# B&R Automation Studio project RTFProj (part 2)

#### measurement_ofScore.c
```c
#include <bur/plctypes.h>
#include <bur/plc.h>
#include <astime.h>
#include <string.h>
#include <math.h>

#ifdef __cplusplus
	extern "C"
	{
#endif
	#include "rp_funcx1.h"
#ifdef __cplusplus
	};
#endif
void initialization(struct measurement_ofScore* m_oS);

void measurement_ofScore(struct measurement_ofScore* m_oS)
{

    if(!m_oS->Enable){
        initialization(m_oS);
    }

    switch(m_oS->Internal.state){
        case 0:
            {
                if(m_oS->Internal.counter <= 0){
                    m_oS->Internal.counter = 0;
                }

                m_oS->Internal.results[0]   = strcmp(m_oS->PLAYER1_NAME, "");
                m_oS->Internal.results[1]   = strcmp(m_oS->PLAYER2_NAME, "");

                if(m_oS->start_measurement == 1 && m_oS->Error == 0){
                    if(m_oS->Internal.results[0] == 0 && m_oS->Internal.results[1] == 0){
                        m_oS->Internal.auxiliary_str[5] = (UDINT) strcpy(m_oS->PLAYER1_NAME,"PLAYER 1");
                        m_oS->Internal.auxiliary_str[6] = (UDINT) strcpy(m_oS->PLAYER2_NAME,"PLAYER 2");
                    }
                    // CPU NAME
                    m_oS->Internal.auxiliary_str[7] = (UDINT) strcpy(m_oS->team_nameCPU,"B&R ROBOT");
                    // HUMAN NAME
                    strcpy(m_oS->Internal.string[5],m_oS->PLAYER1_NAME);
                    strcpy(m_oS->Internal.string[6]," \n \t& \n");
                    strcpy(m_oS->Internal.string[8], m_oS->PLAYER2_NAME);
                    m_oS->Internal.auxiliary_str[8] = (UDINT) strcat(m_oS->Internal.string[5], m_oS->Internal.string[6]);
                    strcpy(m_oS->Internal.string[7], m_oS->Internal.string[5]);
                    m_oS->Internal.auxiliary_str[9] = (UDINT) strcat(m_oS->Internal.string[7], m_oS->Internal.string[8]);
                    m_oS->Internal.auxiliary_str[10] = (UDINT) strcpy(m_oS->team_nameHUM,m_oS->Internal.auxiliary_str[9]);
                    // CHANGE STATE
                    m_oS->Internal.state = 1;
                }else if(m_oS->Error == 1){
                    m_oS->Internal.state = 5;
                }else if(m_oS->pause == 1){
                    m_oS->Internal.before_state = m_oS->Internal.state;
                    m_oS->Internal.state = 6;
                }else{
                    m_oS->Internal.state = 0;
                }
            }
            break;
        case 1:
            {
                if(m_oS->sens_wicket_CPU == 1){
                    m_oS->count_goals_CPU++;
                    m_oS->sens_wicket_CPU = 0;
                }

                if(m_oS->sens_wicket_HUM == 1){
                    m_oS->count_goals_HUM++;
                    m_oS->sens_wicket_HUM = 0;
                }

                if((m_oS->count_goals_HUM - m_oS->count_goals_CPU) == 0){
                    m_oS->probability_CPU = 50;
                    m_oS->probability_HUM = 50;
                }else if((m_oS->count_goals_HUM - m_oS->count_goals_CPU) < 0){
                    if(fabs((m_oS->count_goals_HUM - m_oS->count_goals_CPU)) <= 5){
                        m_oS->probability_CPU = 50 + fabs((m_oS->count_goals_HUM - m_oS->count_goals_CPU))*10;
                        m_oS->probability_HUM = 100 - m_oS->probability_CPU;
                    }else{
                        m_oS->probability_CPU = 100;
                        m_oS->probability_HUM = 0;
                    }
                }else{
                    if(fabs((m_oS->count_goals_HUM - m_oS->count_goals_CPU)) <= 5){
                        m_oS->probability_HUM = 50 + fabs((m_oS->count_goals_HUM - m_oS->count_goals_CPU))*10;
                        m_oS->probability_CPU = 100 - m_oS->probability_HUM;
                    }else{
                        m_oS->probability_HUM = 100;
                        m_oS->probability_CPU = 0;
                    }
                }
				if(((m_oS->count_goals_CPU + m_oS->count_goals_HUM) == 10) && m_oS->Error == 0){
					if(m_oS->count_goals_CPU > m_oS->count_goals_HUM){
						m_oS->Internal.WINNER++;
					}else if(m_oS->count_goals_CPU == m_oS->count_goals_HUM){
						m_oS->Internal.DRAW++;
					}else if(m_oS->count_goals_CPU < m_oS->count_goals_HUM){
						m_oS->Internal.LOSE++;
					}
					// change state
					m_oS->Internal.state             = 2;
					m_oS->Internal.write_matchInfo   = 1;
				}else if(m_oS->exit_game == 1 ){
                    m_oS->Internal.state = 3;
                }else if(m_oS->restart_measurement == 1){
                    m_oS->Internal.state = 4;
                }else if(m_oS->Error == 1){
                    m_oS->Internal.state = 5;
                }else if(m_oS->pause == 1){
                    m_oS->Internal.before_state = m_oS->Internal.state;
                    m_oS->Internal.state = 6;
                }else{
                    m_oS->Internal.state = 1;
                }

            }
            break;
        case 2:
            {
                if(m_oS->Internal.write_matchInfo == 1){
                    // call FB : Get time and date
                    m_oS->Internal.UtcDTStructureGetTime_1.enable = 1;
                    m_oS->Internal.UtcDTStructureGetTime_1.pDTStructure = (UDINT) &m_oS->Internal.DTStruct;
                    UtcDTStructureGetTime(&m_oS->Internal.UtcDTStructureGetTime_1);
                    ascDTStructure((UDINT) &m_oS->Internal.DTStruct, (UDINT) &m_oS->Internal.string[0], m_oS->Internal.length);
                    // write time and date into the variable
                    m_oS->Internal.auxiliary_str[0] = (UDINT) strcpy(m_oS->match_informations.date[m_oS->Internal.counter],m_oS->Internal.string[0]);
                    // write score
                    m_oS->match_informations.score_CPU[m_oS->Internal.counter] = m_oS->count_goals_CPU;
                    m_oS->match_informations.score_HUM[m_oS->Internal.counter] = m_oS->count_goals_HUM;
                    // write name of B&R team
                    m_oS->Internal.auxiliary_str[1] = (UDINT) strcpy(m_oS->match_informations.team_name_CPU[m_oS->Internal.counter],"B&R ROBOT");
                    // write names of both players
                    strcpy(m_oS->Internal.string[1],m_oS->PLAYER1_NAME);
                    strcpy(m_oS->Internal.string[2]," & ");
                    strcpy(m_oS->Internal.string[4], m_oS->PLAYER2_NAME);
                    m_oS->Internal.auxiliary_str[2] = (UDINT) strcat(m_oS->Internal.string[1], m_oS->Internal.string[2]);
                    strcpy(m_oS->Internal.string[3], m_oS->Internal.string[1]);
                    m_oS->Internal.auxiliary_str[3] = (UDINT) strcat(m_oS->Internal.string[3], m_oS->Internal.string[4]);
                    m_oS->Internal.auxiliary_str[4] = (UDINT) strcpy(m_oS->match_informations.team_name_HUM[m_oS->Internal.counter],m_oS->Internal.auxiliary_str[3]);

                    m_oS->Internal.counter++;
                    m_oS->Internal.write_matchInfo = 0;
                }

                if(m_oS->exit_game == 1){
                    m_oS->Internal.state = 3;
                }else if(m_oS->restart_measurement == 1){
                    m_oS->Internal.state = 4;
                }else if(m_oS->Error == 1){
                    m_oS->Internal.state = 5;
                }else if(m_oS->pause == 1){
                    m_oS->Internal.before_state = m_oS->Internal.state;
                    m_oS->Internal.state = 6;
                }else{
                    m_oS->Internal.state = 2;
                }
            }
            break;
        case 3:
            {
                // exit game
                m_oS->start_measurement   = 0;
                m_oS->exit_game           = 0;
                m_oS->restart_measurement = 0;
                m_oS->count_goals_CPU     = 0;
                m_oS->count_goals_HUM     = 0;

                m_oS->Internal.e_r_str[0] = (UDINT) strcpy(m_oS->PLAYER1_NAME,"");
                m_oS->Internal.e_r_str[1] = (UDINT) strcpy(m_oS->PLAYER2_NAME,"");

                if(m_oS->Error == 1){
                    m_oS->Internal.state = 5;
                }else if(m_oS->pause == 1){
                    m_oS->Internal.before_state = m_oS->Internal.state;
                    m_oS->Internal.state = 6;
                }else{
                    m_oS->Internal.state = 0;
                }
            }
            break;
        case 4:
            {
                // restart game
                m_oS->start_measurement   = 0;
                m_oS->exit_game           = 0;
                m_oS->restart_measurement = 0;
                m_oS->count_goals_CPU     = 0;
                m_oS->count_goals_HUM     = 0;

                m_oS->Internal.e_r_str[2] = (UDINT) strcpy(m_oS->PLAYER1_NAME,m_oS->PLAYER1_NAME);
                m_oS->Internal.e_r_str[3] = (UDINT) strcpy(m_oS->PLAYER2_NAME,m_oS->PLAYER2_NAME);

                if(m_oS->Error == 1){
                    m_oS->Internal.state = 5;
                }else if(m_oS->pause == 1){
                    m_oS->Internal.before_state = m_oS->Internal.state;
                    m_oS->Internal.state = 6;
                }else{
                    m_oS->Internal.state = 1;
                }
            }
            break;
        case 5:
            {
                // error state
                if(m_oS->Error == 0){
                    m_oS->Internal.state = 3;
                }else if(m_oS->pause == 1){
                    m_oS->Internal.before_state = m_oS->Internal.state;
                    m_oS->Internal.state = 6;
                }
            }
            break;
        case 6:
            {
                // pause
                if(m_oS->Error == 1){
                    m_oS->Internal.state = 5;
                }else if(m_oS->pause == 0){
                    m_oS->Internal.state = m_oS->Internal.before_state;
                }
            }
            break;
    }// end switch

}// end fucntion

void initialization(struct measurement_ofScore* m_oS){
    m_oS->Internal.state             = 0;
    m_oS->Internal.e_r_str[0]        = 0;
    m_oS->Internal.e_r_str[1]        = 0;
    m_oS->Internal.e_r_str[2]        = 0;
    m_oS->Internal.e_r_str[3]        = 0;
    m_oS->Internal.auxiliary_str[0]  = 0;
    m_oS->Internal.auxiliary_str[1]  = 0;
    m_oS->Internal.auxiliary_str[2]  = 0;
    m_oS->Internal.auxiliary_str[3]  = 0;
    m_oS->Internal.auxiliary_str[4]  = 0;
    m_oS->Internal.auxiliary_str[5]  = 0;
    m_oS->Internal.auxiliary_str[6]  = 0;
    m_oS->Internal.auxiliary_str[7]  = 0;
    m_oS->Internal.auxiliary_str[8]  = 0;
    m_oS->Internal.auxiliary_str[9]  = 0;
    m_oS->Internal.auxiliary_str[10] = 0;
    m_oS->Internal.counter           = 0;
    m_oS->Internal.length            = 25;
    m_oS->Internal.write_matchInfo   = 0;
    m_oS->Internal.results[0]        = 0;
    m_oS->Internal.results[1]        = 0;
	m_oS->Internal.before_state      = 0;
	m_oS->Internal.WINNER			 = 0;
	m_oS->Internal.DRAW			     = 0;
	m_oS->Internal.LOSE				 = 0;
    m_oS->count_goals_CPU            = 0;
    m_oS->count_goals_HUM            = 0;
    m_oS->sens_wicket_HUM            = 0;
    m_oS->restart_measurement        = 0;
    m_oS->pause                      = 0;
    m_oS->exit_game                  = 0;
    m_oS->start_measurement          = 0;
    m_oS->probability_CPU            = 50;
    m_oS->probability_HUM            = 50;
}// end function
```

#### start_linearAxis.c
```c
#include <bur/plctypes.h>
#include <stdio.h>
#include <stdlib.h>
#include <MpAxis.h>

#ifdef __cplusplus
	extern "C"
	{
#endif
	#include "rp_funcx1.h"
#ifdef __cplusplus
	};
#endif
void initialization_sla(struct start_linearAxis* s_la);

void start_linearAxis(struct start_linearAxis* s_la)
{
	if(!s_la->Enable){
		initialization_sla(s_la);
	}

	switch(s_la->Internal.state){
		case 0:
			{
				s_la->Internal.before_state     = s_la->Internal.state;

				if(s_la->start_btn == 1){
					// adjustment parameters -> axis
					s_la->axis_param->Home.Mode 				  = mpAXIS_HOME_MODE_BLOCK_TORQUE;
					s_la->axis_param->Home.Position 		  	  = s_la->max_leftPosition;
					s_la->axis_param->Home.StartVelocity   		  = s_la->velocity;
					s_la->axis_param->Home.HomingVelocity  		  = s_la->velocity;
					s_la->axis_param->Home.Acceleration    		  = 200000;
					s_la->axis_param->Home.StartDirection  		  = mpAXIS_HOME_DIR_POSITIVE;
					s_la->axis_param->Home.HomingDirection 		  = mpAXIS_HOME_DIR_NEGATIVE;
					s_la->axis_param->Home.TorqueLimit	 		  = 0.02;
					s_la->axis_param->Home.PositionErrorStopLimit = s_la->max_leftPosition + 10;
					// reset output
					s_la->succesfully = 0;
					if(s_la->axis_name->Error == 1 || s_la->axis_name->StatusID != 0){
						s_la->axis_name->ErrorReset = 0;
						if(s_la->axis_name->ErrorReset == 0){
							s_la->Internal.state = 10;
						}
					}else{
						if(s_la->start_btn == 1){
							s_la->Internal.state = 1;
						}
					}
				}
			}
			break;
		case 1:
			{
				s_la->Internal.before_state = s_la->Internal.state;
				// power on -> axis
				s_la->axis_name->Power = 1;

				if(s_la->axis_name->Error == 1 || s_la->axis_name->StatusID != 0){
					s_la->axis_name->ErrorReset = 0;
					if(s_la->axis_name->ErrorReset == 0){
						s_la->Internal.state = 10;
					}
				}else{
					if(s_la->axis_name->PowerOn == 1){
						s_la->Internal.state = 2;
					}
				}
			}
			break;
		case 2:
			{
				s_la->Internal.before_state = s_la->Internal.state;
				// update -> axis
				s_la->axis_name->Update = 1;

				if(s_la->axis_name->Error == 1 || s_la->axis_name->StatusID != 0){
					s_la->axis_name->ErrorReset = 0;
					if(s_la->axis_name->ErrorReset == 0){
						s_la->Internal.state = 10;
					}
				}else{
					if(s_la->axis_name->UpdateDone == 1){
						s_la->axis_name->Update = 0;
						if(s_la->axis_name->UpdateDone == 0){
							s_la->Internal.state 	= 3;
						}
					}
				}
			}
		case 3:
			{
				s_la->Internal.before_state = s_la->Internal.state;
				// home -> axis
				s_la->axis_name->Home = 1;

				if(s_la->axis_name->Error == 1 || s_la->axis_name->StatusID != 0){
					s_la->axis_name->ErrorReset = 0;
					if(s_la->axis_name->ErrorReset == 0){
						s_la->Internal.state = 10;
					}
				}else{
					if(s_la->axis_name->IsHomed == 1){
						s_la->axis_name->Home = 0;
						s_la->succesfully     = 1;
						s_la->Internal.state  = 0;
					}
				}
			}
			break;
		case 10:
			{
				s_la->axis_name->ErrorReset = 1;

				if(s_la->axis_name->Error == 1 || s_la->axis_name->StatusID != 0){
					s_la->Internal.state = 10;
				}else{
					s_la->axis_name->ErrorReset = 0;
					s_la->Internal.state 		= s_la->Internal.before_state;
				}
			}
			break;
	}// end switch
}// end function

void initialization_sla(struct start_linearAxis* s_la)
{
	s_la->Internal.state 		= 0;
	s_la->Internal.before_state = 0;
	s_la->start_btn				= 0;
	s_la->succesfully     		= 0;
}// end function
```

#### start_virtualAxis.c
```c
#include <bur/plctypes.h>
#include <stdio.h>
#include <stdlib.h>
#include <MpAxis.h>

#ifdef __cplusplus
	extern "C"
	{
#endif
	#include "rp_funcx1.h"
#ifdef __cplusplus
	};
#endif
void initialization_sva(struct start_virtualAxis* s_va);

void start_virtualAxis(struct start_virtualAxis* s_va)
{
	if(!s_va->Enable){
		initialization_sra(s_va);
	}

	switch(s_va->Internal.state){
		case 0:
			{
				s_va->Internal.before_state     = s_va->Internal.state;

				if(s_va->start_btn == 1){
					// reset output {virtual}
					s_va->succesfully = 0;
					if(s_va->axis_name->Error == 1 || s_va->axis_name->StatusID != 0){
						s_va->axis_name->ErrorReset = 0;
						if(s_va->axis_name->ErrorReset == 0){
							s_va->Internal.state = 10;
						}
					}else{
						if(s_va->start_btn == 1){
							s_va->Internal.state = 1;
						}
					}
				}
			}
			break;
		case 1:
			{
				s_va->Internal.before_state = s_va->Internal.state;
				// power on -> axis
				s_va->axis_name->Power = 1;

				if(s_va->axis_name->Error == 1 || s_va->axis_name->StatusID != 0){
					s_va->axis_name->ErrorReset = 0;
					if(s_va->axis_name->ErrorReset == 0){
						s_va->Internal.state = 10;
					}
				}else{
					if(s_va->axis_name->PowerOn == 1){
						s_va->Internal.state = 2;
					}
				}
			}
			break;
		case 2:
			{
				s_va->Internal.before_state = s_va->Internal.state;
				// home -> axis
				s_va->axis_name->Home = 1;

				if(s_va->axis_name->Error == 1 || s_va->axis_name->StatusID != 0){
					s_va->axis_name->ErrorReset = 0;
					if(s_va->axis_name->ErrorReset == 0){
						s_va->Internal.state = 10;
					}
				}else{
					if(s_va->axis_name->IsHomed == 1){
						s_va->axis_name->Home = 0;
						s_va->Internal.state  = 3;
					}
				}
			}
			break;
		case 3:
			{
				s_va->Internal.before_state = s_va->Internal.state;

				if(s_va->axis_name->Error == 1 || s_va->axis_name->StatusID != 0){
					s_va->axis_name->ErrorReset = 0;
					if(s_va->axis_name->ErrorReset == 0){
						s_va->Internal.state = 10;
					}
				}else{
					s_va->succesfully	 = 1;
					s_va->Internal.state = 0;
				}
			}
			break;
		case 10:
			{
				s_va->axis_name->ErrorReset = 1;

				if(s_va->axis_name->Error == 1 || s_va->axis_name->StatusID != 0){
					s_va->Internal.state = 10;
				}else{
					s_va->axis_name->ErrorReset = 0;
					s_va->Internal.state 		= s_va->Internal.before_state;
				}
			}
			break;
	}// end switch
}// end function

void initialization_sva(struct start_virtualAxis* s_va)
{
	s_va->Internal.state 		= 0;
	s_va->Internal.before_state = 0;
	s_va->start_btn				= 0;
	s_va->succesfully     		= 0;
}// end function
```

#### start_rotaryAxis.c
```c
#include <bur/plctypes.h>
#include <stdio.h>
#include <stdlib.h>
#include <MpAxis.h>

#ifdef __cplusplus
	extern "C"
	{
#endif
	#include "rp_funcx1.h"
#ifdef __cplusplus
	};
#endif
void initialization_sra(struct start_rotaryAxis* s_ra);

void start_rotaryAxis(struct start_rotaryAxis* s_ra)
{
	if(!s_ra->Enable){
		initialization_sra(s_ra);
	}

	switch(s_ra->Internal.state){
		case 0:
			{
				s_ra->Internal.before_state     = s_ra->Internal.state;

				if(s_ra->start_btn == 1){
					// adjust param -> axis
					// move position
					s_ra->axis_param->Acceleration = 3969754;
					s_ra->axis_param->Deceleration = 3969754;
					s_ra->axis_param->Velocity     = 1000;
					s_ra->axis_param->Position 	   = 0;
					// home
					s_ra->axis_param->Home.Position = s_ra->value_ofRotatation;
					// reset output
					s_ra->succesfully = 0;
					if(s_ra->axis_name->Error == 1 || s_ra->axis_name->StatusID != 0){
						s_ra->axis_name->ErrorReset = 0;
						if(s_ra->axis_name->ErrorReset == 0){
							s_ra->Internal.state = 10;
						}
					}else{
						if(s_ra->start_btn == 1){
							s_ra->Internal.state = 1;
						}
					}
				}
			}
			break;
		case 1:
			{
				s_ra->Internal.before_state = s_ra->Internal.state;
				// power on -> axis
				s_ra->axis_name->Power = 1;

				if(s_ra->axis_name->Error == 1 || s_ra->axis_name->StatusID != 0){
					s_ra->axis_name->ErrorReset = 0;
					if(s_ra->axis_name->ErrorReset == 0){
						s_ra->Internal.state = 10;
					}
				}else{
					if(s_ra->axis_name->PowerOn == 1){
						s_ra->Internal.state = 2;
					}
				}
			}
			break;
		case 2:
			{
				s_ra->Internal.before_state = s_ra->Internal.state;
				// update -> axis
				s_ra->axis_name->Update = 1;

				if(s_ra->axis_name->Error == 1 || s_ra->axis_name->StatusID != 0){
					s_ra->axis_name->ErrorReset = 0;
					if(s_ra->axis_name->ErrorReset == 0){
						s_ra->Internal.state = 10;
					}
				}else{
					if(s_ra->axis_name->UpdateDone == 1){
						s_ra->axis_name->Update = 0;
						if(s_ra->axis_name->Update == 0){
							s_ra->Internal.state = 3;
						}
					}
				}
			}
		case 3:
			{
				s_ra->Internal.before_state = s_ra->Internal.state;
				// home -> axis
				s_ra->axis_name->Home = 1;

				if(s_ra->axis_name->Error == 1 || s_ra->axis_name->StatusID != 0){
					s_ra->axis_name->ErrorReset = 0;
					if(s_ra->axis_name->ErrorReset == 0){
						s_ra->Internal.state = 10;
					}
				}else{
					if(s_ra->axis_name->IsHomed == 1){
						s_ra->axis_name->Home = 0;
						s_ra->Internal.state  = 4;
					}
				}
			}
			break;
		case 4:
			{
				s_ra->Internal.before_state = s_ra->Internal.state;
				// move absolute -> axis
				s_ra->axis_name->MoveAbsolute = 1;

				if(s_ra->axis_name->Error == 1 || s_ra->axis_name->StatusID != 0){
					s_ra->axis_name->ErrorReset = 0;
					if(s_ra->axis_name->ErrorReset == 0){
						s_ra->Internal.state = 10;
					}
				}else{
					if(s_ra->axis_name->InPosition == 1){
						s_ra->axis_name->MoveAbsolute = 0;

						if(s_ra->axis_name->MoveAbsolute == 0){
							s_ra->succesfully	 = 1;
							s_ra->Internal.state = 0;
						}
					}
				}
			}
			break;
		case 10:
			{
				s_ra->axis_name->ErrorReset = 1;

				if(s_ra->axis_name->Error == 1 || s_ra->axis_name->StatusID != 0){
					s_ra->Internal.state = 10;
				}else{
					s_ra->axis_name->ErrorReset = 0;
					s_ra->Internal.state 		= s_ra->Internal.before_state;
				}
			}
			break;
	}// end switch
}// end function

void initialization_sra(struct start_rotaryAxis* s_ra)
{
	s_ra->Internal.state 		= 0;
	s_ra->Internal.before_state = 0;
	s_ra->start_btn				= 0;
	s_ra->succesfully     		= 0;
}// end function
```

#### err_detection.c
```c
#include <bur/plctypes.h>
#ifdef __cplusplus
	extern "C"
	{
#endif
	#include "rp_funcx1.h"
#ifdef __cplusplus
	};
#endif

void err_detection(struct err_detection* e_d)
{
	USINT i, count_err;
	// initialization variables
	count_err = 0;
	// output
	e_d->err_detect = 0;

	for(i = 0; i < (int)(sizeof(e_d->rotary_ERR)/sizeof(e_d->rotary_ERR[0])); i++){
		if((e_d->rotary_ERR[i] == 1 || e_d->linear_ERR[i]) == 1){
			count_err = 1;
		}
	}

	if(count_err == 0){
		e_d->err_detect = 0;
	}else{
		e_d->err_detect = 1;
	}
}
```

#### control_temperature.c
```c
#include <bur/plctypes.h>
#ifdef __cplusplus
	extern "C"
	{
#endif
	#include "rp_funcx1.h"
#ifdef __cplusplus
	};
#endif

void control_temperature(struct control_temperature* c_t)
{
	USINT i;
	USINT MAX_TEMPERATURE_ROTARY = 100, MAX_TEMPERATURE_LINEAR = 100;

	for(i = 0; i < (int)(sizeof(c_t->temperature_rotary)/sizeof(c_t->temperature_rotary[0])); i++){
		if(c_t->temperature_rotary[i] >= MAX_TEMPERATURE_ROTARY){
			c_t->high_temp_rotary[i] = 1;
		}else{
			c_t->high_temp_rotary[i] = 0;
		}

		if(c_t->temperature_linear[i] >= MAX_TEMPERATURE_LINEAR){
			c_t->high_temp_linear[i] 	 = 1;
			c_t->start_cooling_linear[i] = 1;
		}else{
			c_t->high_temp_linear[i] 	 = 0;
			c_t->start_cooling_linear[i] = 0;
		}
	}
}
```

#### ball_shooting.c
```c
#include <bur/plctypes.h>
#include <stdio.h>
#include <stdlib.h>
#include <MpAxis.h>

#ifdef __cplusplus
	extern "C"
	{
#endif
	#include "rp_funcx1.h"
#ifdef __cplusplus
	};
#endif
void init_ball_shooting(struct ball_shooting* b_s);
void ball_shooting(struct ball_shooting* b_s)
{
	if(b_s->Enable == 0){
		init_ball_shooting(&b_s);
	}

	switch(b_s->Internal.state){
		case 0:
			{
				if(b_s->start_shoot == 1){
					// initialization parameters of axes for shooting ball
					b_s->rotary_axes->CyclicPosition = 1;
					b_s->rotary_axes->Position		 = -500;
					b_s->rotary_axes->Velocity 		 = 63000;

					// change state
					b_s->Internal.state = 1;
				}
			}
			break;
		case 1:
			{
				if(b_s->rotary_axes->Info.SlavePosition == b_s->rotary_axes->Position){
					// second position
					b_s->rotary_axes->Position	= 500;
					if(b_s->rotary_axes->Info.SlavePosition == 500){
						b_s->Internal.state = 2;
					}
				}
			}
			break;
		case 2:
			{
				if(b_s->rotary_axes->Info.SlavePosition == b_s->rotary_axes->Position){
					// second position
					b_s->rotary_axes->Position	= -250;

					if(b_s->rotary_axes->Info.SlavePosition == -250){
						b_s->successfully = 1;
						if(b_s->successfully == 1){
							b_s->Internal.state = 0;
						}
					}
				}

			}
			break;
	}// end switch
}// end function

void init_ball_shooting(struct ball_shooting* b_s)
{
	b_s->Internal.state = 0;
	b_s->successfully   = 0;
	b_s->start_shoot    = 0;
}
```

#### turn_position.c
```c
#include <bur/plctypes.h>
#include <stdio.h>
#include <stdlib.h>
#include <MpAxis.h>

#ifdef __cplusplus
	extern "C"
	{
#endif
	#include "rp_funcx1.h"
#ifdef __cplusplus
	};
#endif
void initial_turn_pos(struct turn_position* t_p);
void turn_position(struct turn_position* t_p)
{
	if(t_p->Enable == 0){
		initial_turn_pos(&t_p);
	}

	switch(t_p->Internal.state){
		case 0:
			{
				// parameters of move
				t_p->Internal.distance_ofMovePos  = 100 + 170 + 80 + 150;
				t_p->Internal.distance_ofMoveNeg  = (-1)*t_p->Internal.distance_ofMovePos;
				// velocity
				t_p->rotary_axes->Velocity 		= 1500;
				t_p->linear_axes->Velocity 		= 500;
				// initialization parameters
				t_p->Internal.max_pos_ofAxes[0] = 800;
				t_p->Internal.max_pos_ofAxes[1] = 1030;
				t_p->Internal.max_pos_ofAxes[2] = 520;
				t_p->Internal.max_pos_ofAxes[3] = 830;

				t_p->Internal.min_pos_ofAxes[0] = -910;
				t_p->Internal.min_pos_ofAxes[1] = -930;
				t_p->Internal.min_pos_ofAxes[2] = -500;
				t_p->Internal.min_pos_ofAxes[3] = -770;

				// start function
				if(t_p->start_turn == 1){
					t_p->successfully = 0;
					if(t_p->successfully == 0){
						// first position
						t_p->rotary_axes->Position = 500;
						if((t_p->linear_axes->Info.SlavePosition + t_p->Internal.distance_ofMovePos) > t_p->Internal.max_pos_ofAxes[t_p->index_ofAxis]){
							t_p->Internal.auxiliary_move_pos = t_p->linear_axes->Info.SlavePosition;
							t_p->linear_axes->Position = t_p->linear_axes->Info.SlavePosition + t_p->Internal.distance_ofMoveNeg;
						}else if((t_p->linear_axes->Info.SlavePosition + t_p->Internal.distance_ofMovePos) < t_p->Internal.min_pos_ofAxes[t_p->index_ofAxis]){
							t_p->Internal.auxiliary_move_pos = t_p->linear_axes->Info.SlavePosition;
							t_p->linear_axes->Position = t_p->linear_axes->Info.SlavePosition + t_p->Internal.distance_ofMovePos;
						}else{
							t_p->Internal.auxiliary_move_pos = t_p->linear_axes->Info.SlavePosition;
							t_p->linear_axes->Position = t_p->linear_axes->Info.SlavePosition + t_p->Internal.distance_ofMovePos;
						}
						// change state
						t_p->Internal.state = 1;

					}
				}
			}
			break;
		case 1:
			{

				if((t_p->rotary_axes->Position == t_p->rotary_axes->Info.SlavePosition) &&(t_p->linear_axes->Position == t_p->linear_axes->Info.SlavePosition)){
					t_p->rotary_axes->Position = -500;
					t_p->Internal.state = 2;
				}

			}
			break;
		case 2:
			{
				if((t_p->rotary_axes->Position == t_p->rotary_axes->Info.SlavePosition) &&(t_p->linear_axes->Position == t_p->linear_axes->Info.SlavePosition)){
					// initial position
					t_p->linear_axes->Position = t_p->Internal.distance_ofMoveNeg;
					t_p->rotary_axes->Position = -250;
					// change state
					t_p->Internal.state = 3;
				}

			}
			break;
		case 3:
			{
				if((t_p->rotary_axes->Position == t_p->rotary_axes->Info.SlavePosition) &&(t_p->linear_axes->Position == t_p->linear_axes->Info.SlavePosition)){
					t_p->successfully = 1;
					t_p->Internal.state = 0;
				}

			}
			break;
	}// end switch
}// end function

void initial_turn_pos(struct turn_position* t_p)
{
	t_p->Internal.state = 0;
	t_p->successfully   = 0;
	t_p->start_turn		= 0;
}
```

#### check_attack_mode.c
```c
#include <bur/plctypes.h>
#ifdef __cplusplus
	extern "C"
	{
#endif
	#include "rp_funcx1.h"
#ifdef __cplusplus
	};
#endif

void check_attack_mode(struct check_attack_mode* ch_aM)
{
	struct calculation_posDummies calculation_posDummies_0;
	struct detect_axisNumber detect_axisNumber_0;
	struct choose_attack_mode choose_attack_mode_0;
	INT behind_position, before_position;
	USINT i_chp, i_aM, stand_mode;
	REAL max_pos[4], min_pos[4];

	max_pos[0] = 800;
	max_pos[1] = 1060;
	max_pos[2] = 550;
	max_pos[3] = 860;

	min_pos[0] = -910;
	min_pos[1] = -960;
	min_pos[2] = -530;
	min_pos[3] = -800;

	for(i_chp = 0; i_chp < (int)(sizeof(ch_aM->act_displacement_cpu)/sizeof(ch_aM->act_displacement_cpu[0])); i_chp++){
		calculation_posDummies_0.displacement[i_chp] = ch_aM->act_displacement_cpu[i_chp];
		calculation_posDummies_0.max_disp[i_chp]	 = max_pos[i_chp];
		calculation_posDummies_0.min_disp[i_chp]	 = min_pos[i_chp];
	}

	calculation_posDummies(&calculation_posDummies_0);

	detect_axisNumber_0.ball1_x = ch_aM->ball1_x;
	detect_axisNumber_0.ball2_x = ch_aM->ball2_x;
	detect_axisNumber(&detect_axisNumber_0);

	if(detect_axisNumber_0.axis_number != 10){
		if(ch_aM->angle_ofRotation[detect_axisNumber_0.axis_number] > 0){
			// stand before the ball
			behind_position = -90;
			before_position = 90;
			stand_mode		= 1;
		}else{
			// stand behind the ball
			behind_position = -200; // -170
			before_position = 350;  // 320
			stand_mode		= 2;
		}

		for(i_aM = 0; i_aM < (int)(sizeof(calculation_posDummies_0.actual_positionsOfDummies)/sizeof(calculation_posDummies_0.actual_positionsOfDummies[0])); i_aM++){
			choose_attack_mode_0.actual_positionsOfDummies[i_aM] = calculation_posDummies_0.actual_positionsOfDummies[i_aM];
		}
		choose_attack_mode_0.ball1_x 		 = ch_aM->ball1_x;
		choose_attack_mode_0.ball1_y 		 = ch_aM->ball1_y;
		choose_attack_mode_0.ball2_x 		 = ch_aM->ball2_x;
		choose_attack_mode_0.ball2_y 		 = ch_aM->ball2_y;
		choose_attack_mode_0.axis_number 	 = detect_axisNumber_0.axis_number;
		choose_attack_mode_0.before_position = before_position;
		choose_attack_mode_0.behind_position = behind_position;
		choose_attack_mode(&choose_attack_mode_0);

		if((choose_attack_mode_0.mode == 1) && (stand_mode == 1)){
			ch_aM->attack_mode = 1; // attack mode If ball is behind of dummy
		}else if((choose_attack_mode_0.mode == 1) && (stand_mode == 2)){
			ch_aM->attack_mode = 2; // attack mode If ball is before of dummy
		}else{
			ch_aM->attack_mode = 0; // If ball it isn't near of dummy
		}

		ch_aM->index_ofAxis = detect_axisNumber_0.axis_number;
	}else{
		ch_aM->attack_mode  = 0;
		ch_aM->index_ofAxis = 0;
	}

}

void detect_axisNumber(struct detect_axisNumber* d_aN)
{
	INT x_posOfD[4];
	REAL x_pos[2];
	USINT i_dAn, a_n[2];

	x_posOfD[0] = 800;
	x_posOfD[1] = 2300;
	x_posOfD[2] = 5300;
	x_posOfD[3] = 8300;

	x_pos[0] = d_aN->ball1_x;
	x_pos[1] = d_aN->ball2_x;

	for(i_dAn = 0; i_dAn < (int)(sizeof(x_pos)/sizeof(x_pos[0])); i_dAn++){
		if(x_pos[i_dAn] >= (x_posOfD[3] - 90)){
			a_n[i_dAn] = 3;
		}else if((x_pos[i_dAn] >= (x_posOfD[2] - 90)) && (x_pos[i_dAn] <= (x_posOfD[3] - 90))){
			a_n[i_dAn] = 2;
		}else if((x_pos[i_dAn] >= (x_posOfD[1] - 90)) && (x_pos[i_dAn] <= (x_posOfD[2] - 90))){
			a_n[i_dAn] = 1;
		}else if((x_pos[i_dAn] >= (x_posOfD[0] - 90)) && (x_pos[i_dAn] <= (x_posOfD[1] - 90))){
			a_n[i_dAn] = 0;
		}else{
			a_n[i_dAn] = 10;
		}

	}

	if((a_n[0] == a_n[1]) || isnan(x_pos[1])){
		d_aN->axis_number = a_n[0];
	}else{
		d_aN->axis_number = a_n[1];
	}
}

void choose_attack_mode(struct choose_attack_mode* ch_aMode)
{
	USINT aux_mode;
	USINT i_df, i_md, i_fw;
	INT x_posOfD[4];
	REAL gk_pos, df_pos[2], md_pos[5], fw_pos[3];

	// auxiliary mode
	aux_mode = 0;
	// initial x pos of axes CPU
	x_posOfD[0] = 800;
	x_posOfD[1] = 2300;
	x_posOfD[2] = 5300;
	x_posOfD[3] = 8300;

	// goalkeeper
	gk_pos = ch_aMode->actual_positionsOfDummies[0];
	// defender
	df_pos[0] = ch_aMode->actual_positionsOfDummies[1];
	df_pos[1] = ch_aMode->actual_positionsOfDummies[2];
	// midfielder
	md_pos[0] = ch_aMode->actual_positionsOfDummies[3];
	md_pos[1] = ch_aMode->actual_positionsOfDummies[4];
	md_pos[2] = ch_aMode->actual_positionsOfDummies[5];
	md_pos[3] = ch_aMode->actual_positionsOfDummies[6];
	md_pos[4] = ch_aMode->actual_positionsOfDummies[7];
	// forward
	fw_pos[0] = ch_aMode->actual_positionsOfDummies[8];
	fw_pos[1] = ch_aMode->actual_positionsOfDummies[9];
	fw_pos[2] = ch_aMode->actual_positionsOfDummies[10];

	switch(ch_aMode->axis_number){
		case 0:
			{
				if((((ch_aMode->ball1_x <= (x_posOfD[ch_aMode->axis_number] + ch_aMode->before_position))
					&& (ch_aMode->ball1_x >= (x_posOfD[ch_aMode->axis_number] + ch_aMode->behind_position)))
					|| ((ch_aMode->ball2_x <= (x_posOfD[ch_aMode->axis_number] + ch_aMode->before_position))
					&& (ch_aMode->ball2_x >= (x_posOfD[ch_aMode->axis_number] + ch_aMode->behind_position))))
					&& ((ch_aMode->ball1_y <= (gk_pos + 150)) && (ch_aMode->ball1_y >= (gk_pos - 150))
					|| ((ch_aMode->ball2_y <= (gk_pos + 150)) && (ch_aMode->ball2_y >= (gk_pos - 150))))){
					aux_mode = 1;
				}else{
					aux_mode = 0;
				}
			}
			break;
		case 1:
			{
				for(i_df = 0; i_df < (int)(sizeof(df_pos)/sizeof(df_pos[0])); i_df++){
					if((((ch_aMode->ball1_x <= (x_posOfD[ch_aMode->axis_number] + ch_aMode->before_position))
						&& (ch_aMode->ball1_x >= (x_posOfD[ch_aMode->axis_number] + ch_aMode->behind_position)))
						|| ((ch_aMode->ball2_x <= (x_posOfD[ch_aMode->axis_number] + ch_aMode->before_position))
						&& (ch_aMode->ball2_x >= (x_posOfD[ch_aMode->axis_number] + ch_aMode->behind_position))))
						&& ((ch_aMode->ball1_y <= (df_pos[i_df] + 150)) && (ch_aMode->ball1_y >= (df_pos[i_df] - 150))
						|| ((ch_aMode->ball2_y <= (df_pos[i_df] + 150)) && (ch_aMode->ball2_y >= (df_pos[i_df] - 150))))){
						aux_mode = 1;
					}
				}
			}
			break;
		case 2:
			{
				for(i_md = 0; i_md < (int)(sizeof(md_pos)/sizeof(md_pos[0])); i_md++){
					if((((ch_aMode->ball1_x <= (x_posOfD[ch_aMode->axis_number] + ch_aMode->before_position))
						&& (ch_aMode->ball1_x >= (x_posOfD[ch_aMode->axis_number] + ch_aMode->behind_position)))
						|| ((ch_aMode->ball2_x <= (x_posOfD[ch_aMode->axis_number] + ch_aMode->before_position))
						&& (ch_aMode->ball2_x >= (x_posOfD[ch_aMode->axis_number] + ch_aMode->behind_position))))
						&& ((ch_aMode->ball1_y <= (md_pos[i_md] + 150)) && (ch_aMode->ball1_y >= (md_pos[i_md] - 150))
						|| ((ch_aMode->ball2_y <= (md_pos[i_md] + 150)) && (ch_aMode->ball2_y >= (md_pos[i_md] - 150))))){
						aux_mode = 1;
					}
				}
			}
			break;
		case 3:
			{
				for(i_fw = 0; i_fw < (int)(sizeof(fw_pos)/sizeof(fw_pos[0])); i_fw++){
					if((((ch_aMode->ball1_x <= (x_posOfD[ch_aMode->axis_number] + ch_aMode->before_position))
						&& (ch_aMode->ball1_x >= (x_posOfD[ch_aMode->axis_number] + ch_aMode->behind_position)))
						|| ((ch_aMode->ball2_x <= (x_posOfD[ch_aMode->axis_number] + ch_aMode->before_position))
						&& (ch_aMode->ball2_x >= (x_posOfD[ch_aMode->axis_number] + ch_aMode->behind_position))))
						&& ((ch_aMode->ball1_y <= (fw_pos[i_fw] + 150)) && (ch_aMode->ball1_y >= (fw_pos[i_fw] - 150))
						|| ((ch_aMode->ball2_y <= (fw_pos[i_fw] + 150)) && (ch_aMode->ball2_y >= (fw_pos[i_fw] - 150))))){
						aux_mode = 1;
					}
				}
			}
			break;
	}// end switch

	if(aux_mode == 1){
		ch_aMode->mode = aux_mode;
	}else{
		ch_aMode->mode = 0;
	}
}
```

#### axes_control.c
```c
#include <bur/plctypes.h>
#include <stdio.h>
#include <stdlib.h>
#include <MpAxis.h>

#ifdef __cplusplus
	extern "C"
	{
#endif
	#include "rp_funcx1.h"
#ifdef __cplusplus
	};
#endif
void init_control_axis(struct axes_control* a_c);

void axes_control(struct axes_control* a_c)
{

	if(!a_c->Enable){
		init_control_axis(&a_c);
	}

	switch(a_c->Internal.state){
		case 0:
			{
				a_c->Internal.before_state = 0;

				if(a_c->start_move == 1){
					a_c->successfully = 0;

					if(a_c->successfully == 0){
						if(((a_c->rotary_axis_cyclic->Error == 1 && a_c->rotary_axis_cyclic->StatusID != 0) || (a_c->linear_axis_cyclic->Error == 1 && a_c->linear_axis_cyclic->StatusID != 0))
						|| (a_c->rotary_axis_cyclic->CommandAborted == 1 || a_c->linear_axis_cyclic->CommandAborted == 1)){
							// cyclic position -> off
							a_c->linear_axis_cyclic->CyclicPosition = 0;
							a_c->rotary_axis_cyclic->CyclicPosition = 0;
							if(a_c->linear_axis_cyclic->CyclicPosition == 0 && a_c->rotary_axis_cyclic->CyclicPosition == 0){
								// go to error state
								a_c->Internal.state = 10;
							}
						}else{
							// start cyclic position
							a_c->linear_axis_cyclic->CyclicPosition = 1;
							a_c->rotary_axis_cyclic->CyclicPosition = 1;
							// go to next state
							a_c->Internal.state = 1;
						}
					}else if(((a_c->rotary_axis_cyclic->Error == 1 && a_c->rotary_axis_cyclic->StatusID != 0) || (a_c->linear_axis_cyclic->Error == 1 && a_c->linear_axis_cyclic->StatusID != 0))
					|| (a_c->rotary_axis_cyclic->CommandAborted == 1 || a_c->linear_axis_cyclic->CommandAborted == 1)){
						// cyclic position -> off
						a_c->linear_axis_cyclic->CyclicPosition = 0;
						a_c->rotary_axis_cyclic->CyclicPosition = 0;
						if(a_c->linear_axis_cyclic->CyclicPosition == 0 && a_c->rotary_axis_cyclic->CyclicPosition == 0){
							// go to error state
							a_c->Internal.state = 10;
						}
					}
				}
			}
			break;
		case 1:
			{
				a_c->Internal.before_state = 1;

				if(a_c->linear_axis_param->Acceleration == a_c->linear_param.acceleration && a_c->linear_axis_cyclic->Velocity == a_c->linear_param.velocity){
					if(a_c->rotary_axis_param->Acceleration == a_c->rotary_param.acceleration && a_c->rotary_axis_cyclic->Velocity == a_c->rotary_param.velocity){
						if(((a_c->rotary_axis_cyclic->Error == 1 && a_c->rotary_axis_cyclic->StatusID != 0) || (a_c->linear_axis_cyclic->Error == 1 && a_c->linear_axis_cyclic->StatusID != 0))
						|| (a_c->rotary_axis_cyclic->CommandAborted == 1 || a_c->linear_axis_cyclic->CommandAborted == 1)){
							// cyclic position -> off
							a_c->linear_axis_cyclic->CyclicPosition = 0;
							a_c->rotary_axis_cyclic->CyclicPosition = 0;
							if(a_c->linear_axis_cyclic->CyclicPosition == 0 && a_c->rotary_axis_cyclic->CyclicPosition == 0){
								// go to error state
								a_c->Internal.state = 10;
							}
						}else{
							a_c->Internal.state = 2;
						}
					}else{
						if(((a_c->rotary_axis_cyclic->Error == 1 && a_c->rotary_axis_cyclic->StatusID != 0) || (a_c->linear_axis_cyclic->Error == 1 && a_c->linear_axis_cyclic->StatusID != 0))
						|| (a_c->rotary_axis_cyclic->CommandAborted == 1 || a_c->linear_axis_cyclic->CommandAborted == 1)){
							// cyclic position -> off
							a_c->linear_axis_cyclic->CyclicPosition = 0;
							a_c->rotary_axis_cyclic->CyclicPosition = 0;
							if(a_c->linear_axis_cyclic->CyclicPosition == 0 && a_c->rotary_axis_cyclic->CyclicPosition == 0){
								// go to error state
								a_c->Internal.state = 10;
							}
						}else{
							a_c->Internal.state = 3;
						}
					}
				}else{
					if(a_c->rotary_axis_param->Acceleration == a_c->rotary_param.acceleration && a_c->rotary_axis_cyclic->Velocity == a_c->rotary_param.velocity){
						if(((a_c->rotary_axis_cyclic->Error == 1 && a_c->rotary_axis_cyclic->StatusID != 0) || (a_c->linear_axis_cyclic->Error == 1 && a_c->linear_axis_cyclic->StatusID != 0))
						|| (a_c->rotary_axis_cyclic->CommandAborted == 1 || a_c->linear_axis_cyclic->CommandAborted == 1)){
							// cyclic position -> off
							a_c->linear_axis_cyclic->CyclicPosition = 0;
							a_c->rotary_axis_cyclic->CyclicPosition = 0;
							if(a_c->linear_axis_cyclic->CyclicPosition == 0 && a_c->rotary_axis_cyclic->CyclicPosition == 0){
								// go to error state
								a_c->Internal.state = 10;
							}
						}else{
							a_c->Internal.state = 4;
						}
					}else{
						if(((a_c->rotary_axis_cyclic->Error == 1 && a_c->rotary_axis_cyclic->StatusID != 0) || (a_c->linear_axis_cyclic->Error == 1 && a_c->linear_axis_cyclic->StatusID != 0))
						|| (a_c->rotary_axis_cyclic->CommandAborted == 1 || a_c->linear_axis_cyclic->CommandAborted == 1)){
							// cyclic position -> off
							a_c->linear_axis_cyclic->CyclicPosition = 0;
							a_c->rotary_axis_cyclic->CyclicPosition = 0;
							if(a_c->linear_axis_cyclic->CyclicPosition == 0 && a_c->rotary_axis_cyclic->CyclicPosition == 0){
								// go to error state
								a_c->Internal.state = 10;
							}
						}else{
							a_c->Internal.state = 5;
						}
					}
				}
			}
			break;
		case 2:
			{
				a_c->Internal.before_state = 2;

				// linear axis param cyclic
				a_c->linear_axis_cyclic->Position 				= a_c->linear_param.displacement;
				// rotary axis param cyclic
				a_c->rotary_axis_cyclic->Position 				= a_c->rotary_param.displacement;

				if(((a_c->rotary_axis_cyclic->Error == 1 && a_c->rotary_axis_cyclic->StatusID != 0) || (a_c->linear_axis_cyclic->Error == 1 && a_c->linear_axis_cyclic->StatusID != 0))
				|| (a_c->rotary_axis_cyclic->CommandAborted == 1 || a_c->linear_axis_cyclic->CommandAborted == 1)){
					// cyclic position -> off
					a_c->linear_axis_cyclic->CyclicPosition = 0;
					a_c->rotary_axis_cyclic->CyclicPosition = 0;
					if(a_c->linear_axis_cyclic->CyclicPosition == 0 && a_c->rotary_axis_cyclic->CyclicPosition == 0){
						// go to error state
						a_c->Internal.state = 10;
					}
				}else{
					a_c->Internal.state = 6;
				}
			}
			break;
		case 3:
			{
				a_c->Internal.before_state = 3;
				// turn off
				a_c->rotary_axis_cyclic->CyclicPosition = 0;

				if(a_c->rotary_axis_cyclic->CyclicPosition == 0){
					// linear axis param cyclic
					a_c->linear_axis_cyclic->Velocity   			= a_c->linear_param.velocity;
					a_c->linear_axis_cyclic->Position 				= a_c->linear_param.displacement;
					// rotary axis param
					a_c->rotary_axis_param->Acceleration		    = a_c->rotary_param.acceleration;
					a_c->rotary_axis_param->Deceleration			= a_c->rotary_param.deceleration;
					// rotary axis param cyclic
					a_c->rotary_axis_cyclic->Velocity   			= a_c->rotary_param.velocity;
					a_c->rotary_axis_cyclic->Position 				= a_c->rotary_param.displacement;

					// update parameters
					a_c->rotary_axis_cyclic->Update = 1;

					if(((a_c->rotary_axis_cyclic->Error == 1 && a_c->rotary_axis_cyclic->StatusID != 0) || (a_c->linear_axis_cyclic->Error == 1 && a_c->linear_axis_cyclic->StatusID != 0))
					 || (a_c->rotary_axis_cyclic->CommandAborted == 1 || a_c->linear_axis_cyclic->CommandAborted == 1)){
						// cyclic position -> off
						a_c->linear_axis_cyclic->CyclicPosition = 0;
						a_c->rotary_axis_cyclic->CyclicPosition = 0;
						if(a_c->linear_axis_cyclic->CyclicPosition == 0 && a_c->rotary_axis_cyclic->CyclicPosition == 0){
							// go to error state
							a_c->Internal.state = 10;
						}
					}else{
						if(a_c->rotary_axis_cyclic->UpdateDone == 1){
							a_c->rotary_axis_cyclic->Update = 0;
							if(a_c->rotary_axis_cyclic->Update == 0){
								// turn on
								a_c->rotary_axis_cyclic->CyclicPosition = 1;
								if(a_c->rotary_axis_cyclic->CyclicPosition == 1){
									a_c->Internal.state = 6;
								}
							}
						}
					}
				}
			}
			break;
		case 4:
			{
				a_c->Internal.before_state = 4;

				// turn off
				a_c->linear_axis_cyclic->CyclicPosition = 0;

				if(a_c->linear_axis_cyclic->CyclicPosition == 0){
					// linear axis param
					a_c->linear_axis_param->Acceleration		    = a_c->linear_param.acceleration;
					a_c->linear_axis_param->Deceleration			= a_c->linear_param.deceleration;
					// linear axis param cyclic
					a_c->linear_axis_cyclic->Velocity   			= a_c->linear_param.velocity;
					a_c->linear_axis_cyclic->Position 				= a_c->linear_param.displacement;
					// rotary axis param cyclic
					a_c->rotary_axis_cyclic->Velocity   			= a_c->rotary_param.velocity;
					a_c->rotary_axis_cyclic->Position 				= a_c->rotary_param.displacement;

					// update parameters
					a_c->linear_axis_cyclic->Update = 1;

					if(((a_c->rotary_axis_cyclic->Error == 1 && a_c->rotary_axis_cyclic->StatusID != 0) || (a_c->linear_axis_cyclic->Error == 1 && a_c->linear_axis_cyclic->StatusID != 0))
					|| (a_c->rotary_axis_cyclic->CommandAborted == 1 || a_c->linear_axis_cyclic->CommandAborted == 1)){
						// cyclic position -> off
						a_c->linear_axis_cyclic->CyclicPosition = 0;
						a_c->rotary_axis_cyclic->CyclicPosition = 0;
						if(a_c->linear_axis_cyclic->CyclicPosition == 0 && a_c->rotary_axis_cyclic->CyclicPosition == 0){
							// go to error state
							a_c->Internal.state = 10;
						}
					}else{
						if(a_c->linear_axis_cyclic->UpdateDone == 1){
							a_c->linear_axis_cyclic->Update = 0;
							if(a_c->linear_axis_cyclic->Update == 0){
								// turn on
								a_c->linear_axis_cyclic->CyclicPosition = 1;
								if(a_c->linear_axis_cyclic->CyclicPosition == 1){
									a_c->Internal.state = 6;
								}
							}
						}
					}
				}
			}
			break;
		case 5:
			{
				a_c->Internal.before_state = 5;

				// turn off
				a_c->linear_axis_cyclic->CyclicPosition = 0;
				a_c->rotary_axis_cyclic->CyclicPosition = 0;

				if(a_c->linear_axis_cyclic->CyclicPosition == 0 && a_c->rotary_axis_cyclic->CyclicPosition == 0){
					// linear axis param
					a_c->linear_axis_param->Acceleration		    = a_c->linear_param.acceleration;
					a_c->linear_axis_param->Deceleration			= a_c->linear_param.deceleration;
					// linear axis param cyclic
					a_c->linear_axis_cyclic->Velocity   			= a_c->linear_param.velocity;
					a_c->linear_axis_cyclic->Position 				= a_c->linear_param.displacement;
					// rotary axis param
					a_c->rotary_axis_param->Acceleration		    = a_c->rotary_param.acceleration;
					a_c->rotary_axis_param->Deceleration			= a_c->rotary_param.deceleration;
					// rotary axis param cyclic
					a_c->rotary_axis_cyclic->Velocity   			= a_c->rotary_param.velocity;
					a_c->rotary_axis_cyclic->Position 				= a_c->rotary_param.displacement;

					// update parameters
					a_c->linear_axis_cyclic->Update = 1;
					a_c->rotary_axis_cyclic->Update = 1;

					if(((a_c->rotary_axis_cyclic->Error == 1 && a_c->rotary_axis_cyclic->StatusID != 0) || (a_c->linear_axis_cyclic->Error == 1 && a_c->linear_axis_cyclic->StatusID != 0))
					|| (a_c->rotary_axis_cyclic->CommandAborted == 1 || a_c->linear_axis_cyclic->CommandAborted == 1)){
						// cyclic position -> off
						a_c->linear_axis_cyclic->CyclicPosition = 0;
						a_c->rotary_axis_cyclic->CyclicPosition = 0;
						if(a_c->linear_axis_cyclic->CyclicPosition == 0 && a_c->rotary_axis_cyclic->CyclicPosition == 0){
							// go to error state
							a_c->Internal.state = 10;
						}
					}else{
						if(a_c->linear_axis_cyclic->UpdateDone == 1 && a_c->rotary_axis_cyclic->UpdateDone == 1){
							a_c->linear_axis_cyclic->Update = 0;
							a_c->rotary_axis_cyclic->Update = 0;
							if(a_c->linear_axis_cyclic->Update == 0 && a_c->rotary_axis_cyclic->Update == 0){
								// turn on
								a_c->linear_axis_cyclic->CyclicPosition = 1;
								a_c->rotary_axis_cyclic->CyclicPosition = 1;
								if(a_c->linear_axis_cyclic->CyclicPosition == 1 && a_c->rotary_axis_cyclic->CyclicPosition == 1){
									a_c->Internal.state = 6;
								}
							}
						}
					}
				}
			}
			break;
		case 6:
			{
				a_c->Internal.before_state = 6;

				if(((a_c->rotary_axis_cyclic->Error == 1 && a_c->rotary_axis_cyclic->StatusID != 0) || (a_c->linear_axis_cyclic->Error == 1 && a_c->linear_axis_cyclic->StatusID != 0))
				|| (a_c->rotary_axis_cyclic->CommandAborted == 1 || a_c->linear_axis_cyclic->CommandAborted == 1)){
					// cyclic position -> off
					a_c->linear_axis_cyclic->CyclicPosition = 0;
					a_c->rotary_axis_cyclic->CyclicPosition = 0;
					if(a_c->linear_axis_cyclic->CyclicPosition == 0 && a_c->rotary_axis_cyclic->CyclicPosition == 0){
						// go to error state
						a_c->Internal.state = 10;
					}
				}else{
					a_c->successfully = 1;

					if(a_c->successfully == 1){
						a_c->Internal.state = 0;
					}
				}
			}
			break;
		case 10:
			{
				// error reset -> on
				a_c->rotary_axis_cyclic->ErrorReset = 1;
				a_c->linear_axis_cyclic->ErrorReset = 1;

				if((a_c->rotary_axis_cyclic->Error == 0 && a_c->linear_axis_cyclic->Error == 0 && a_c->rotary_axis_cyclic->StatusID == 0 && a_c->linear_axis_cyclic->StatusID == 0)
				&& (a_c->rotary_axis_cyclic->CommandAborted == 0 && a_c->linear_axis_cyclic->CommandAborted == 0)){
					// error reset -> off
					a_c->rotary_axis_cyclic->ErrorReset = 0;
					a_c->linear_axis_cyclic->ErrorReset = 0;
					// cyclic position -> on
					a_c->linear_axis_cyclic->CyclicPosition = 1;
					a_c->rotary_axis_cyclic->CyclicPosition = 1;

					if(a_c->rotary_axis_cyclic->ErrorReset == 0 && a_c->linear_axis_cyclic->ErrorReset == 0){
						a_c->Internal.state = a_c->Internal.before_state;
					}
				}

			}
			break;
	}// end switch

}// end function

void init_control_axis(struct axes_control* a_c)
{
	a_c->Internal.state 	   = 0;
	a_c->Internal.before_state = 0;
	a_c->successfully 		   = 0;
}
```

#### powerOn_axes.c - not listed in the package file held
```c
#include <bur/plctypes.h>
#include <stdio.h>
#include <stdlib.h>
#include <MpAxis.h>

#ifdef __cplusplus
	extern "C"
	{
#endif
	#include "rp_funcx1.h"
#ifdef __cplusplus
	};
#endif
void initialization_pO_a(struct powerOn_axes* pO_a);

void powerOn_axes(struct powerOn_axes* pO_a)
{
	if(!pO_a->start_btn){
		initialization_pO_a(pO_a);
	}

	switch(pO_a->Internal.state){
		case 0:
			{
				pO_a->Internal.before_state     = pO_a->Internal.state;

				if(pO_a->axis_name_R->Error == 1 || pO_a->axis_name_R->StatusID != 0 || pO_a->axis_name_L->Error == 1 || pO_a->axis_name_L->StatusID != 0){
					pO_a->Internal.state = 10;
				}else{
					if(pO_a->start_btn == 1){
						pO_a->Internal.state = 1;
					}
				}
			}
			break;
		case 1:
			{
				pO_a->Internal.before_state = pO_a->Internal.state;
				// power on -> axis
				pO_a->axis_name_R->Power = 1;
				pO_a->axis_name_L->Power = 1;

				if(pO_a->axis_name_R->PowerOn == 1 && pO_a->axis_name_L->PowerOn == 1){
					pO_a->succesfully = 1;
				}else if(pO_a->axis_name_R->Error == 1 || pO_a->axis_name_L->StatusID != 0){
					pO_a->Internal.state = 10;
				}else{
					pO_a->Internal.state = pO_a->Internal.before_state;
				}
			}
			break;
		case 10:
			{
				pO_a->axis_name_R->ErrorReset = 1;
				pO_a->axis_name_L->ErrorReset = 1;

			if(pO_a->axis_name_R->Error == 1 || pO_a->axis_name_R->StatusID != 0 || pO_a->axis_name_L->Error == 1 || pO_a->axis_name_L->StatusID != 0){
					pO_a->Internal.state = 10;
				}else{
					pO_a->axis_name_R->ErrorReset = 0;
					pO_a->axis_name_L->ErrorReset = 0;
					pO_a->Internal.state 		= pO_a->Internal.before_state;
				}
			}
			break;
	}// end switch
}// end function

void initialization_pO_a(struct powerOn_axes* pO_a)
{
	pO_a->Internal.state 		= 0;
	pO_a->Internal.before_state = 0;
	pO_a->start_btn				= 0;
	pO_a->succesfully     		= 0;
}// end function
```

### Package Logical/Libraries/RO_LB_ScoreDetection - Lubo and Radek Library for detection of score.

### Library Logical/Libraries/RO_LB_ScoreDetection/GoalKeeper (ANSIC)
Depends on: standard

#### GoalKeeper.c
```c
#include <bur/plctypes.h>

#ifdef _DEFAULT_INCLUDES
#include <AsDefault.h>
#endif

void GoalKeeper(struct GoalKeeper *inst){

	if (inst->enable){
		if (!inst->Internal.init){
			inst->Internal.DisableTimer1.PT = inst->Internal.DisableTimer2.PT = 100;
			inst->Internal.init = 1;
		}

		if (!inst->DI9371.ModuleOk)
			inst->status = ERR_DI_NOTFOUND;
		else{
			inst->status = ERR_OK;

			TON_10ms(&inst->Internal.DisableTimer1);

			if ((inst->Internal.DisableTimer1.IN == 1) && (inst->Internal.DisableTimer1.Q))
				inst->Internal.DisableTimer1.IN = 0;
			else if ((!inst->DI9371.DigitalInput_1) && (!inst->isGoal1) && (!inst->Internal.DisableTimer1.IN)) {
				inst->isGoal1 = 1;
				inst->Internal.DisableTimer1.IN = 1;
			}
			else inst->isGoal1 = 0;

			TON_10ms(&inst->Internal.DisableTimer2);

			if ((inst->Internal.DisableTimer2.IN == 1) && (inst->Internal.DisableTimer2.Q))
				inst->Internal.DisableTimer2.IN = 0;
			else if ((!inst->DI9371.DigitalInput_2) && (!inst->isGoal2) && (!inst->Internal.DisableTimer2.IN)) {
				inst->isGoal2 = 1;
				inst->Internal.DisableTimer2.IN = 1;
			}
			else inst->isGoal2 = 0;
		}
	}
	else
		inst->status = ERR_FUB_ENABLE_FALSE;
}
```

#### Types.typ - Exported data types
```iecst
TYPE
	DI9371_type : 	STRUCT
		ModuleOk : BOOL;
		DigitalInput_1 : BOOL;
		DigitalInput_2 : BOOL;
	END_STRUCT;
	InternalG_type : 	STRUCT
		init : BOOL;
		DisableTimer1 : TON_10ms;
		DisableTimer2 : TON_10ms;
	END_STRUCT;
END_TYPE
```

#### Constants.var - Exported constants
```iecst
VAR CONSTANT
	ERR_DI_NOTFOUND : UDINT := 45813;
END_VAR
```

#### GoalKeeper.fun - Exported functions and function blocks
```iecst
FUNCTION_BLOCK GoalKeeper
	VAR_INPUT
		enable : BOOL;
		DI9371 : DI9371_type;
	END_VAR
	VAR_OUTPUT
		status : UINT;
		isGoal1 : BOOL;
		isGoal2 : BOOL;
	END_VAR
	VAR
		Internal : InternalG_type;
	END_VAR
END_FUNCTION_BLOCK
```

### Library Logical/Libraries/IecCheck (IEC)
Depends on: sys_lib, AsBrStr

### Library Logical/Libraries/RO_Sensors (IEC)

#### Types.typ - Exported data types
```iecst
TYPE
	PositionStatus :
		(
		PosCalcPos, (*1*)
		PosInitial
		);
	Stuct_OptSensInternal : 	STRUCT
		TransConstant : ARRAY[0..3]OF INT;
		MaxPosHum : ARRAY[0..3]OF INT := [1025,1700,675,975];
		MinPosHum : ARRAY[0..3]OF INT := [-1025,-1700,-675,-975];
		RefPosHum : ARRAY[0..3]OF INT := [4(0)];
		MaxPosSens : ARRAY[0..3]OF INT := [31406,31852,32495,31208];
		MinPosSens : ARRAY[0..3]OF INT := [13652,6831,23895,12431];
		RefPosSens : ARRAY[0..3]OF INT := [22798,18167,28195,21044];
		Index : ARRAY[0..5]OF USINT;
		DR_ReflexSensStatus_0 : DetectionRotation;
		DP_Figure_0 : DetPos_Figure;
		MinAccDiff : INT := 100;
		MaxAccDiff : ARRAY[0..3]OF INT := [4(100)];
		CurrentPosition : ARRAY[0..3]OF INT;
	END_STRUCT;
	Stuct_RexlSensInternal : 	STRUCT
		ActReflexSensStatusRS : ARRAY[0..3]OF BOOL;
		ErrorStatusRS : ARRAY[0..3]OF BOOL;
		ExternalReflexSensStatusRS : ARRAY[0..3]OF BOOL;
		ReflexSensStatusRS : ARRAY[0..3]OF BOOL;
		IndexR : ARRAY[0..1]OF USINT;
	END_STRUCT;
	Struct_OptSensFigInternal : 	STRUCT
		MaxPosHumDP : ARRAY[0..3]OF INT;
		MinPosHumDP : ARRAY[0..3]OF INT;
		DispAxisDP : ARRAY[0..10]OF INT := [0,-1200,1200,-2400,-1200,0,1200,2400,-2100,0,2100];
		CurrentPosition : ARRAY[0..10]OF INT;
		Index : ARRAY[0..2]OF USINT;
	END_STRUCT;
	Struct_CorrectionFun : 	STRUCT
		CorrectionPosition : ARRAY[0..3]OF INT;
		FundamentalVal : FundamentalType;
		ComputedPosition : ARRAY[0..3]OF ComputedPosType := [(Comp:=[-1130,-1056,-930,-789,-661,-498,-356,-221,-84,51,167,260,343,444,528,593,678,748,835,908,985,1021,13(5000)]),(Comp:=[-1618,-1517,-1419,-1296,-1187,-1077,-970,-863,-758,-656,-543,-454,-337,-236,-141,-36,65,163,271,381,490,606,693,791,903,1000,1120,1218,1343,1440,1541,1625,1744,1875,1945]),(Comp:=[-634,-526,-397,-259,-158,-39,55,177,278,368,479,582,698,777,21(5000)]),(Comp:=[-954,-834,-714,-620,-488,-397,-266,-163,-47,73,155,261,344,431,532,618,719,836,931,1051,1119,14(5000)])];
		RealPositionMeasured : ARRAY[0..3]OF MeasPosMesType := [(Meas:=[-1025,-925,-825,-725,-625,-525,-425,-325,-225,-125,-25,75,175,275,375,475,575,675,775,875,975,1025,13(5000)]),(Meas:=[-1700,-1600,-1500,-1400,-1300,-1200,-1100,-1000,-900,-800,-700,-600,-500,-400,-300,-200,-100,0,100,200,300,400,500,600,700,800,900,1000,1100,1200,1300,1400,1500,1600,1700]),(Meas:=[-675,-575,-475,-375,-275,-175,-75,25,125,225,325,425,525,675,21(5000)]),(Meas:=[-975,-875,-775,-675,-575,-475,-375,-275,-175,-75,25,125,225,325,425,525,625,725,825,925,975,14(5000)])];
		Index : IndexType;
		DifferenceYi : DifferenceType;
	END_STRUCT;
	DifferenceType : 	STRUCT
		Y0 : ARRAY[0..34]OF INT; (*21 valid members of the field*)
		Y1 : ARRAY[0..34]OF INT; (*34 valid members of the field*)
		Y2 : ARRAY[0..34]OF INT; (*13 valid members of the field*)
		Y3 : ARRAY[0..34]OF INT; (*20 valid members of the field*)
	END_STRUCT;
	RealPosMesType1 : 	STRUCT
		RealPosAxisGoalkeeper : ARRAY[0..34]OF INT := [-1025,-925,-825,-725,-625,-525,-425,-325,-225,-125,-25,75,175,275,375,475,575,675,775,875,975,1025,13(5000)];
		RealPosAxisDefender : ARRAY[0..34]OF INT := [-1700,-1600,-1500,-1400,-1300,-1200,-1100,-1000,-900,-800,-700,-600,-500,-400,-300,-200,-100,0,100,200,300,400,500,600,700,800,900,1000,1100,1200,1300,1400,1500,1600,1700];
		RealPosAxisMidfielder : ARRAY[0..34]OF INT := [-675,-575,-475,-375,-275,-175,-75,25,125,225,325,425,525,675,21(5000)];
		RealPosAxisAttaker : ARRAY[0..34]OF INT := [-975,-875,-775,-675,-575,-475,-375,-275,-175,-75,25,125,225,325,425,525,625,725,825,925,975,14(5000)];
	END_STRUCT;
	ComputedPosType1 : 	STRUCT
		CompPosAxisGoalkeeper : ARRAY[0..34]OF INT := [-1130,-1056,-930,-789,-661,-498,-356,-221,-84,51,167,260,343,444,528,593,678,748,835,908,985,1021,13(5000)];
		CompPosAxisDefender : ARRAY[0..34]OF INT := [-1618,-1517,-1419,-1296,-1187,-1077,-970,-863,-758,-656,-543,-454,-337,-236,-141,-36,65,163,271,381,490,606,693,791,903,1000,1120,1218,1343,1440,1541,1625,1744,1875,1945];
		CompPosAxisMidfielder : ARRAY[0..34]OF INT := [-634,-526,-397,-259,-158,-39,55,177,278,368,479,582,698,777,21(5000)];
		CompPosAxisAttaker : ARRAY[0..34]OF INT := [-954,-834,-714,-620,-488,-397,-266,-163,-47,73,155,261,344,431,532,618,719,836,931,1051,1119,14(5000)];
	END_STRUCT;
	MeasPosMesType : 	STRUCT
		Meas : ARRAY[0..34]OF INT;
	END_STRUCT;
	ComputedPosType : 	STRUCT
		Comp : ARRAY[0..34]OF INT;
	END_STRUCT;
	IndexType : 	STRUCT
		i0 : INT;
		i1 : INT;
		i2 : INT;
		i3 : INT;
	END_STRUCT;
	FundamentalType : 	STRUCT
		L0 : ARRAY[0..21]OF INT;
		L1 : ARRAY[0..37]OF INT;
		L2 : ARRAY[0..13]OF INT;
		L3 : ARRAY[0..20]OF INT;
	END_STRUCT;
END_TYPE
```

#### RO_Sensors.fun - Exported functions and function blocks
```iecst
FUNCTION_BLOCK DetectionPositionAxis
	VAR_INPUT
		ActPosSens : ARRAY[0..3] OF INT; (*Input value from sensors [SU].*)
		ErrorOptSens : ARRAY[0..3] OF BOOL; (*Error status of optical sensors.*)
		ReflexSensStatus : ARRAY[0..3] OF BOOL; (*Stauts of reflex sensors.*)
	END_VAR
	VAR_OUTPUT
		ActPosHumFig : ARRAY[0..10] OF INT; (*Actual position of every figure of EACH AXIS (displacement of actual position of human axis).*)
		ActPosHumAxis : ARRAY[0..3] OF INT; (*Actual computed value of EACH AXIS with CORRECTIONS.*)
	END_VAR
	VAR
		ActPosHumBasic : ARRAY[0..3] OF INT; (*Value of actual computed value of position of EACH AXIS without CORRECTIONS.*)
		CorrectionPos : Struct_CorrectionFun;
	END_VAR
	VAR_OUTPUT
		ExternalReflexSensStatus : ARRAY[0..3] OF BOOL; (*Status of reflex sensor, which determines two rotation positions.*)
	END_VAR
	VAR
		InternalPos : Stuct_OptSensInternal; (*Internal position determine a position one step before an actual state of actual human (figure) axis.*)
	END_VAR
END_FUNCTION_BLOCK

FUNCTION_BLOCK DetectionRotation
	VAR_INPUT
		ErrorReflSensRS : ARRAY[0..3] OF BOOL;
		ReflexSensStatusRS : ARRAY[0..3] OF BOOL;
	END_VAR
	VAR_OUTPUT
		ExternalReflexSensStatusRS : ARRAY[0..3] OF BOOL;
		ActReflRotRS : ARRAY[0..3] OF BOOL;
	END_VAR
	VAR
		InternalRot : Stuct_RexlSensInternal;
	END_VAR
END_FUNCTION_BLOCK

FUNCTION_BLOCK DetPos_Figure
	VAR_INPUT
		ActPosHumAxisDP : ARRAY[0..3] OF INT;
	END_VAR
	VAR_OUTPUT
		ActPosHumFigDP : ARRAY[0..10] OF INT;
	END_VAR
	VAR
		InternalPosFig : Struct_OptSensFigInternal;
	END_VAR
END_FUNCTION_BLOCK
```

#### DetectionRotation.st
```iecst
(* LOGIC PREDICTION OF ROTATION ALL AXES *)
FUNCTION_BLOCK DetectionRotation

	// Checking the status of reflex sensor
	FOR InternalRot.IndexR[0] := 0 TO 3 DO

		// Reflex sensor works & Modul set TRUE to output
		IF (ReflexSensStatusRS[InternalRot.IndexR[0]] = TRUE) AND (ErrorReflSensRS[InternalRot.IndexR[0]] = FALSE) THEN
			ActReflRotRS[InternalRot.IndexR[0]] := ReflexSensStatusRS[InternalRot.IndexR[0]];

		// Reflex sensor works but Modul set FALSE to output
		ELSIF (ReflexSensStatusRS[InternalRot.IndexR[0]] = FALSE) AND (ErrorReflSensRS[InternalRot.IndexR[0]] = FALSE) THEN
				ActReflRotRS[InternalRot.IndexR[0]] := ReflexSensStatusRS[InternalRot.IndexR[0]];

			// Reflex sensor doesn't works
		ELSIF (ErrorReflSensRS[InternalRot.IndexR[0]] = TRUE) THEN
			ActReflRotRS[InternalRot.IndexR[0]] := FALSE;

		// 	Set the status of Actual position of Rotation by the ModulOK status
		ELSE
			ActReflRotRS[InternalRot.IndexR[0]] := ReflexSensStatusRS[InternalRot.IndexR[0]];
		END_IF
	END_FOR

END_FUNCTION_BLOCK
```

#### DetectionPositionAxis.st
```iecst
(* NUMERIC CALCULATION OF POSITION ALL AXES *)
FUNCTION_BLOCK DetectionPositionAxis

	// Calculate a constants
	InternalPos.TransConstant[0] := (InternalPos.MaxPosSens[0]-InternalPos.MinPosSens[0])/(InternalPos.MaxPosHum[0]-InternalPos.MinPosHum[0]);
	InternalPos.TransConstant[1] := (InternalPos.MaxPosSens[1]-InternalPos.MinPosSens[1])/(InternalPos.MaxPosHum[1]-InternalPos.MinPosHum[1]);
	InternalPos.TransConstant[2] := (InternalPos.MaxPosSens[2]-InternalPos.MinPosSens[2])/(InternalPos.MaxPosHum[2]-InternalPos.MinPosHum[2]);
	InternalPos.TransConstant[3] := (InternalPos.MaxPosSens[3]-InternalPos.MinPosSens[3])/(InternalPos.MaxPosHum[3]-InternalPos.MinPosHum[3]);

	// Lagrange polynomal function for CORRECTION of Computed Position Human Axis
(*	// 1.] Calculate a difference of computed value & measured value of position
	FOR CorrectionPos.Index.i0 := 0 TO 21 DO
		CorrectionPos.DifferenceYi.Y0[CorrectionPos.Index.i0] := CorrectionPos.ComputedPosition.CompPosAxisGoalkeeper[CorrectionPos.Index.i0] - CorrectionPos.RealPositionMeasured.RealPosAxisGoalkeeper[CorrectionPos.Index.i0];
	END_FOR;
	FOR CorrectionPos.Index.i1 := 0 TO 34 DO
		CorrectionPos.DifferenceYi.Y1[CorrectionPos.Index.i1] := CorrectionPos.ComputedPosition.CompPosAxisDefender[CorrectionPos.Index.i1] - CorrectionPos.RealPositionMeasured.RealPosAxisDefender[CorrectionPos.Index.i1];
	END_FOR;
	FOR CorrectionPos.Index.i2 := 0 TO 13 DO
		CorrectionPos.DifferenceYi.Y2[CorrectionPos.Index.i2] := CorrectionPos.ComputedPosition.CompPosAxisMidfielder[CorrectionPos.Index.i2] - CorrectionPos.RealPositionMeasured.RealPosAxisMidfielder[CorrectionPos.Index.i2];
	END_FOR;
	FOR CorrectionPos.Index.i3 := 0 TO 20 DO
		CorrectionPos.DifferenceYi.Y3[CorrectionPos.Index.i3] := CorrectionPos.ComputedPosition.CompPosAxisAttaker[CorrectionPos.Index.i3] - CorrectionPos.RealPositionMeasured.RealPosAxisAttaker[CorrectionPos.Index.i3];
	END_FOR;

	// 2.] Calculate a fundamental polynoms for EACH human axis
	FOR CorrectionPos.Index.i0 := 0 TO 21 DO
	CorrectionPos.FundamentalVal.L0[CorrectionPos.Index.i0] := (((ActPosHumBasic[0]-1)*(ActPosHumBasic[0]-2)*(ActPosHumBasic[0]-3))/((CorrectionPos.RealPositionMeasured.RealPosAxisGoalkeeper[CorrectionPos.Index.i0]-1)*(CorrectionPos.RealPositionMeasured.RealPosAxisGoalkeeper[CorrectionPos.Index.i0]-2)*(CorrectionPos.RealPositionMeasured.RealPosAxisGoalkeeper[CorrectionPos.Index.i0]-3)));
	END_FOR;
	FOR CorrectionPos.Index.i1 := 0 TO 34 DO
		CorrectionPos.FundamentalVal.L1[CorrectionPos.Index.i1] := (((ActPosHumBasic[1]-1)*(ActPosHumBasic[1]-2)*(ActPosHumBasic[1]-3))/((CorrectionPos.RealPositionMeasured.RealPosAxisDefender[CorrectionPos.Index.i1]-1)*(CorrectionPos.RealPositionMeasured.RealPosAxisDefender[CorrectionPos.Index.i1]-2)*(CorrectionPos.RealPositionMeasured.RealPosAxisDefender[CorrectionPos.Index.i1]-3)));
	END_FOR;
	FOR CorrectionPos.Index.i2 := 0 TO 13 DO
		CorrectionPos.FundamentalVal.L2[CorrectionPos.Index.i2] := (((ActPosHumBasic[2]-1)*(ActPosHumBasic[2]-2)*(ActPosHumBasic[2]-3))/((CorrectionPos.RealPositionMeasured.RealPosAxisMidfielder[CorrectionPos.Index.i2]-1)*(CorrectionPos.RealPositionMeasured.RealPosAxisMidfielder[CorrectionPos.Index.i2]-2)*(CorrectionPos.RealPositionMeasured.RealPosAxisMidfielder[CorrectionPos.Index.i2]-3)));
	END_FOR;
	FOR CorrectionPos.Index.i3 := 0 TO 20 DO
		CorrectionPos.FundamentalVal.L3[CorrectionPos.Index.i3] := (((ActPosHumBasic[3]-1)*(ActPosHumBasic[3]-2)*(ActPosHumBasic[3]-3))/((CorrectionPos.RealPositionMeasured.RealPosAxisAttaker[CorrectionPos.Index.i3]-1)*(CorrectionPos.RealPositionMeasured.RealPosAxisAttaker[CorrectionPos.Index.i3]-2)*(CorrectionPos.RealPositionMeasured.RealPosAxisAttaker[CorrectionPos.Index.i3]-3)));
	END_FOR;

	// 3.] Calculate a correction polynomal functions
	// Goalkeeper axis
	CorrectionPos.CorrectionPosition[0] := CorrectionPos.DifferenceYi.Y0[0]*CorrectionPos.FundamentalVal.L0[0]+CorrectionPos.DifferenceYi.Y0[1]*CorrectionPos.FundamentalVal.L0[2]+CorrectionPos.DifferenceYi.Y0[3]*CorrectionPos.FundamentalVal.L0[3]+CorrectionPos.DifferenceYi.Y0[4]*CorrectionPos.FundamentalVal.L0[4]+CorrectionPos.DifferenceYi.Y0[5]*CorrectionPos.FundamentalVal.L0[5]+CorrectionPos.DifferenceYi.Y0[6]*CorrectionPos.FundamentalVal.L0[6]+
	CorrectionPos.DifferenceYi.Y0[7]*CorrectionPos.FundamentalVal.L0[7]+CorrectionPos.DifferenceYi.Y0[8]*CorrectionPos.FundamentalVal.L0[8]+CorrectionPos.DifferenceYi.Y0[9]*CorrectionPos.FundamentalVal.L0[9]+CorrectionPos.DifferenceYi.Y0[10]*CorrectionPos.FundamentalVal.L0[10]+CorrectionPos.DifferenceYi.Y0[11]*CorrectionPos.FundamentalVal.L0[11]+CorrectionPos.DifferenceYi.Y0[12]*CorrectionPos.FundamentalVal.L0[12]+CorrectionPos.DifferenceYi.Y0[13]*CorrectionPos.FundamentalVal.L0[13]
	+CorrectionPos.DifferenceYi.Y0[14]*CorrectionPos.FundamentalVal.L0[14]+CorrectionPos.DifferenceYi.Y0[15]*CorrectionPos.FundamentalVal.L0[15]+CorrectionPos.DifferenceYi.Y0[16]*CorrectionPos.FundamentalVal.L0[16]+CorrectionPos.DifferenceYi.Y0[17]*CorrectionPos.FundamentalVal.L0[17]+CorrectionPos.DifferenceYi.Y0[18]*CorrectionPos.FundamentalVal.L0[18]+CorrectionPos.DifferenceYi.Y0[19]*CorrectionPos.FundamentalVal.L0[19]+CorrectionPos.DifferenceYi.Y0[20]*CorrectionPos.FundamentalVal.L0[20]
	+CorrectionPos.DifferenceYi.Y0[21]*CorrectionPos.FundamentalVal.L0[21];
	// Mid-fielder axis
	CorrectionPos.CorrectionPosition[1] := CorrectionPos.DifferenceYi.Y1[0]*CorrectionPos.FundamentalVal.L1[0]+CorrectionPos.DifferenceYi.Y1[1]*CorrectionPos.FundamentalVal.L1[1]+CorrectionPos.DifferenceYi.Y1[2]*CorrectionPos.FundamentalVal.L1[2]+CorrectionPos.DifferenceYi.Y1[3]*CorrectionPos.FundamentalVal.L1[3]+CorrectionPos.DifferenceYi.Y1[4]*CorrectionPos.FundamentalVal.L1[4]+CorrectionPos.DifferenceYi.Y1[5]*CorrectionPos.FundamentalVal.L1[5]
	+CorrectionPos.DifferenceYi.Y1[6]*CorrectionPos.FundamentalVal.L1[6]+CorrectionPos.DifferenceYi.Y1[7]*CorrectionPos.FundamentalVal.L1[7]+CorrectionPos.DifferenceYi.Y1[8]*CorrectionPos.FundamentalVal.L1[8]+CorrectionPos.DifferenceYi.Y1[9]*CorrectionPos.FundamentalVal.L1[9]+CorrectionPos.DifferenceYi.Y1[10]*CorrectionPos.FundamentalVal.L1[10]+CorrectionPos.DifferenceYi.Y1[11]*CorrectionPos.FundamentalVal.L1[11]+CorrectionPos.DifferenceYi.Y1[12]*CorrectionPos.FundamentalVal.L1[12]
	+CorrectionPos.DifferenceYi.Y1[13]*CorrectionPos.FundamentalVal.L1[13]+CorrectionPos.DifferenceYi.Y1[14]*CorrectionPos.FundamentalVal.L1[14]+CorrectionPos.DifferenceYi.Y1[15]*CorrectionPos.FundamentalVal.L1[15]+CorrectionPos.DifferenceYi.Y1[16]*CorrectionPos.FundamentalVal.L1[16]+CorrectionPos.DifferenceYi.Y1[17]*CorrectionPos.FundamentalVal.L1[17]+CorrectionPos.DifferenceYi.Y1[18]*CorrectionPos.FundamentalVal.L1[18]+CorrectionPos.DifferenceYi.Y1[19]*CorrectionPos.FundamentalVal.L1[19]
	+CorrectionPos.DifferenceYi.Y1[20]*CorrectionPos.FundamentalVal.L1[20]+CorrectionPos.DifferenceYi.Y1[21]*CorrectionPos.FundamentalVal.L1[21]+CorrectionPos.DifferenceYi.Y1[22]*CorrectionPos.FundamentalVal.L1[22]+CorrectionPos.DifferenceYi.Y1[23]*CorrectionPos.FundamentalVal.L1[23]+CorrectionPos.DifferenceYi.Y1[24]*CorrectionPos.FundamentalVal.L1[24]+CorrectionPos.DifferenceYi.Y1[25]*CorrectionPos.FundamentalVal.L1[25]+CorrectionPos.DifferenceYi.Y1[26]*CorrectionPos.FundamentalVal.L1[26]
	+CorrectionPos.DifferenceYi.Y1[27]*CorrectionPos.FundamentalVal.L1[27]+CorrectionPos.DifferenceYi.Y1[28]*CorrectionPos.FundamentalVal.L1[28]+CorrectionPos.DifferenceYi.Y1[29]*CorrectionPos.FundamentalVal.L1[29]+CorrectionPos.DifferenceYi.Y1[30]*CorrectionPos.FundamentalVal.L1[30]+CorrectionPos.DifferenceYi.Y1[31]*CorrectionPos.FundamentalVal.L1[31]+CorrectionPos.DifferenceYi.Y1[32]*CorrectionPos.FundamentalVal.L1[32]+CorrectionPos.DifferenceYi.Y1[33]*CorrectionPos.FundamentalVal.L1[33]
	+CorrectionPos.DifferenceYi.Y1[34]*CorrectionPos.FundamentalVal.L1[34];
	// Defender axis
	CorrectionPos.CorrectionPosition[2] := CorrectionPos.DifferenceYi.Y2[0]*CorrectionPos.FundamentalVal.L2[0]+CorrectionPos.DifferenceYi.Y2[1]*CorrectionPos.FundamentalVal.L2[1]+CorrectionPos.DifferenceYi.Y2[2]*CorrectionPos.FundamentalVal.L2[2]+CorrectionPos.DifferenceYi.Y2[3]*CorrectionPos.FundamentalVal.L2[3]+CorrectionPos.DifferenceYi.Y2[4]*CorrectionPos.FundamentalVal.L2[4]+CorrectionPos.DifferenceYi.Y2[5]*CorrectionPos.FundamentalVal.L2[5]
	+CorrectionPos.DifferenceYi.Y2[6]*CorrectionPos.FundamentalVal.L2[6]+CorrectionPos.DifferenceYi.Y2[7]*CorrectionPos.FundamentalVal.L2[7]+CorrectionPos.DifferenceYi.Y2[8]*CorrectionPos.FundamentalVal.L2[8]+CorrectionPos.DifferenceYi.Y2[9]*CorrectionPos.FundamentalVal.L2[9]+CorrectionPos.DifferenceYi.Y2[10]*CorrectionPos.FundamentalVal.L2[10]+CorrectionPos.DifferenceYi.Y2[11]*CorrectionPos.FundamentalVal.L2[11]+CorrectionPos.DifferenceYi.Y2[12]*CorrectionPos.FundamentalVal.L2[12]
	+CorrectionPos.DifferenceYi.Y2[13]*CorrectionPos.FundamentalVal.L2[13];
	// Attacker axis
	CorrectionPos.CorrectionPosition[3] := CorrectionPos.DifferenceYi.Y3[0]*CorrectionPos.FundamentalVal.L3[0]+CorrectionPos.DifferenceYi.Y3[1]*CorrectionPos.FundamentalVal.L3[1]+CorrectionPos.DifferenceYi.Y3[2]*CorrectionPos.FundamentalVal.L3[2]+CorrectionPos.DifferenceYi.Y3[3]*CorrectionPos.FundamentalVal.L3[3]+CorrectionPos.DifferenceYi.Y3[4]*CorrectionPos.FundamentalVal.L3[4]+CorrectionPos.DifferenceYi.Y3[5]*CorrectionPos.FundamentalVal.L3[5]+CorrectionPos.DifferenceYi.Y3[6]*CorrectionPos.FundamentalVal.L3[6]
	+CorrectionPos.DifferenceYi.Y3[7]*CorrectionPos.FundamentalVal.L3[7]+CorrectionPos.DifferenceYi.Y3[8]*CorrectionPos.FundamentalVal.L3[8]+CorrectionPos.DifferenceYi.Y3[9]*CorrectionPos.FundamentalVal.L3[9]+CorrectionPos.DifferenceYi.Y3[10]*CorrectionPos.FundamentalVal.L3[10]+CorrectionPos.DifferenceYi.Y3[11]*CorrectionPos.FundamentalVal.L3[11]+CorrectionPos.DifferenceYi.Y3[12]*CorrectionPos.FundamentalVal.L3[12]+CorrectionPos.DifferenceYi.Y3[13]*CorrectionPos.FundamentalVal.L3[13]
	+CorrectionPos.DifferenceYi.Y3[14]*CorrectionPos.FundamentalVal.L3[14]+CorrectionPos.DifferenceYi.Y3[15]*CorrectionPos.FundamentalVal.L3[15]+CorrectionPos.DifferenceYi.Y3[16]*CorrectionPos.FundamentalVal.L3[16]+CorrectionPos.DifferenceYi.Y3[17]*CorrectionPos.FundamentalVal.L3[17]+CorrectionPos.DifferenceYi.Y3[18]*CorrectionPos.FundamentalVal.L3[18]+CorrectionPos.DifferenceYi.Y3[19]*CorrectionPos.FundamentalVal.L3[19]+CorrectionPos.DifferenceYi.Y3[20]*CorrectionPos.FundamentalVal.L3[20];
	*)
	// Check the status of Reflex sensors if they work well (TRUE = figure block the balon; FALSE = figure open the way)
	FOR InternalPos.Index[1] := 0 TO 3 DO

		InternalPos.DR_ReflexSensStatus_0.ReflexSensStatusRS[InternalPos.Index[1]] := ReflexSensStatus[InternalPos.Index[1]];
	END_FOR;

	// Calling FB DetRot_ModulOK_0
	InternalPos.DR_ReflexSensStatus_0();

	// Calculation state compute an atual value of distance or set the max/min value
	FOR InternalPos.Index[0] := 0 TO 3 DO

		// Set the External ModulOK value for case disfunction of
		ExternalReflexSensStatus[InternalPos.Index[0]] := InternalPos.DR_ReflexSensStatus_0.ExternalReflexSensStatusRS[InternalPos.Index[0]];

		// Optical sensor work well and values are in range and diference is over the minimal limit (compute a position by equation)
		IF (ErrorOptSens[InternalPos.Index[0]] = FALSE) AND ((ActPosSens[InternalPos.Index[0]] < InternalPos.MaxPosSens[InternalPos.Index[0]]) AND (ABS(ActPosSens[InternalPos.Index[0]] - InternalPos.CurrentPosition[InternalPos.Index[0]]) > InternalPos.MaxAccDiff[0])) AND ((ActPosSens[InternalPos.Index[0]] > InternalPos.MinPosSens[InternalPos.Index[0]]) AND (ABS(ActPosSens[InternalPos.Index[0]] - InternalPos.CurrentPosition[InternalPos.Index[0]]) > InternalPos.MaxAccDiff[0])) THEN
			ActPosHumBasic[InternalPos.Index[0]] := InternalPos.RefPosHum[InternalPos.Index[0]] + ((ActPosSens[InternalPos.Index[0]] - InternalPos.RefPosSens[InternalPos.Index[0]]) / InternalPos.TransConstant[InternalPos.Index[0]]); // Value of computed position without a correction

			(*
			// Compute a corrections for actual position
			FOR InternalPos.Index[4] := 0 TO 33 DO
				IF (CorrectionPos.ComputedPosition[InternalPos.Index[0]].Comp[InternalPos.Index[4]] < ActPosHumBasic[InternalPos.Index[0]] < CorrectionPos.ComputedPosition[InternalPos.Index[0]].Comp[InternalPos.Index[4]+1])  THEN
					InternalPos.Index[5] := InternalPos.Index[4];
					EXIT;
				END_IF;
			END_FOR;
			*)
			CorrectionPos.CorrectionPosition[InternalPos.Index[0]] := (((-1)*(CorrectionPos.ComputedPosition[InternalPos.Index[0]].Comp[InternalPos.Index[5]]-CorrectionPos.ComputedPosition[InternalPos.Index[0]].Comp[InternalPos.Index[5]+1])*(CorrectionPos.RealPositionMeasured[InternalPos.Index[0]].Meas[InternalPos.Index[5]]-ActPosHumBasic[InternalPos.Index[0]]))/(CorrectionPos.RealPositionMeasured[InternalPos.Index[0]].Meas[InternalPos.Index[5]]-CorrectionPos.RealPositionMeasured[InternalPos.Index[0]].Meas[InternalPos.Index[5]+1]));

			// Actual position after corrections
			ActPosHumAxis[InternalPos.Index[0]] := 	ActPosHumBasic[InternalPos.Index[0]]; // - CorrectionPos.CorrectionPosition[InternalPos.Index[0]]; // Corrected value of computed position
			InternalPos.CurrentPosition[InternalPos.Index[0]] := ActPosHumAxis[InternalPos.Index[0]]; // Last detected value is safed as previous value for case Error mode of sensor

			// Optical sensor work well and values are in range and diference is in the minimal limit (set the previous value of position)
		ELSIF (ErrorOptSens[InternalPos.Index[0]] = FALSE) AND ((ActPosSens[InternalPos.Index[0]] < InternalPos.MaxPosSens[InternalPos.Index[0]]) AND (ABS(ActPosSens[InternalPos.Index[0]] - InternalPos.CurrentPosition[InternalPos.Index[0]]) < InternalPos.MaxAccDiff[0])) AND ((ActPosSens[InternalPos.Index[0]] > InternalPos.MinPosSens[InternalPos.Index[0]]) AND (ABS(ActPosSens[InternalPos.Index[0]] - InternalPos.CurrentPosition[InternalPos.Index[0]]) < InternalPos.MaxAccDiff[0])) THEN
			ActPosHumAxis[InternalPos.Index[0]]	:= InternalPos.CurrentPosition[InternalPos.Index[0]]; // Previous value of position

		// Optical sensor doesn't work well but values are in range
		ELSIF (ErrorOptSens[InternalPos.Index[0]] = TRUE) AND (ActPosSens[InternalPos.Index[0]] < InternalPos.MaxPosSens[InternalPos.Index[0]]) AND (ActPosSens[InternalPos.Index[0]] > InternalPos.MinPosSens[InternalPos.Index[0]]) THEN
			ActPosHumAxis[InternalPos.Index[0]] := 	InternalPos.CurrentPosition[InternalPos.Index[0]]; // Previous value of position

		// Optical sensor doesn't work well but values are over the maximum range
		ELSIF (ErrorOptSens[InternalPos.Index[0]] = TRUE) AND ((ActPosSens[InternalPos.Index[0]] > 500) OR (ActPosSens[InternalPos.Index[0]] < 8000))THEN
			ActPosHumAxis[InternalPos.Index[0]] := 	InternalPos.CurrentPosition[InternalPos.Index[0]]; // Previous value of position

		// Check if the Optical sensors are switched on (if not, sensored values are in range <-100 ; +100> _ the minimum limit sets InternalPos.MinAccDiff)
		ELSIF (ActPosSens[InternalPos.Index[0]] < InternalPos.MinAccDiff) THEN
			ActPosHumAxis[InternalPos.Index[0]] := 	InternalPos.RefPosHum[InternalPos.Index[0]]; // Due to a optical sensor fail set referent value of position by previous value of position

		// Check if the Reflex sensors doesn't block the ball (if does, the sensing of position is not required _ just a momentary status)
		ELSIF (ExternalReflexSensStatus[InternalPos.Index[0]] = FALSE) THEN
					ActPosHumAxis[InternalPos.Index[0]] := 	InternalPos.CurrentPosition[InternalPos.Index[0]]; // Due to a reflex sensor fail reset the actual value of position to the referent position

			// Actual human position is set as a last
		ELSE
			ActPosHumAxis[InternalPos.Index[0]] := InternalPos.RefPosHum[InternalPos.Index[0]]; // Set referent position in all other cases as default
		END_IF

	END_FOR;

	// Compute the positions all figures of opponent (by calling the function: DetPos_Figure)
	FOR InternalPos.Index[2] := 0 TO 3 DO

		// Set the input values into the function block
		InternalPos.DP_Figure_0.ActPosHumAxisDP[InternalPos.Index[2]] := ActPosHumAxis[InternalPos.Index[2]];

	END_FOR;

	// Call the function block
	InternalPos.DP_Figure_0();
	FOR InternalPos.Index[3] := 0 TO 10 DO

		// Call the output values of position all figures
 		ActPosHumFig[InternalPos.Index[3]] := InternalPos.DP_Figure_0.ActPosHumFigDP[InternalPos.Index[3]];

	END_FOR;

END_FUNCTION_BLOCK

		(* NUMERIC CALCULATION OF POSITION ALL AXES *)
FUNCTION_BLOCK DetPos_Figure

	// Set the value at position of Goalman Axis by the Actual Position of Axis with Displacement of Axis
	IF (ActPosHumAxisDP[0] < InternalPosFig.MaxPosHumDP[0]) AND (ActPosHumAxisDP[0] > InternalPosFig.MinPosHumDP[0]) THEN
		ActPosHumFigDP[0] := ActPosHumAxisDP[0] + InternalPosFig.DispAxisDP[0];
		InternalPosFig.CurrentPosition[0] := ActPosHumFigDP[0];
	//
	ELSIF ActPosHumAxisDP[0] > InternalPosFig.MaxPosHumDP[0] THEN
		ActPosHumFigDP[0] := InternalPosFig.MaxPosHumDP[0];

	//
	ELSIF ActPosHumAxisDP[0] < InternalPosFig.MinPosHumDP[0] THEN
		ActPosHumFigDP[0] := InternalPosFig.MinPosHumDP[0];

	//
	ELSE
		ActPosHumFigDP[0] := ActPosHumAxisDP[0] + InternalPosFig.DispAxisDP[0];
	END_IF

	FOR InternalPosFig.Index[0] := 1 TO 2 DO
		// Set the value at position of Defender Axis by the Actual Position of Axis with Displacement of Axis
		IF (ActPosHumAxisDP[1] < InternalPosFig.MaxPosHumDP[1]) AND (ActPosHumAxisDP[1] > InternalPosFig.MinPosHumDP[1]) THEN
			ActPosHumFigDP[InternalPosFig.Index[0]] := ActPosHumAxisDP[1] + InternalPosFig.DispAxisDP[InternalPosFig.Index[0]];
			InternalPosFig.CurrentPosition[InternalPosFig.Index[0]] := ActPosHumFigDP[InternalPosFig.Index[0]];
		//
		ELSIF ActPosHumAxisDP[1] > InternalPosFig.MaxPosHumDP[1] THEN
			ActPosHumFigDP[InternalPosFig.Index[0]] := InternalPosFig.MaxPosHumDP[1] + InternalPosFig.DispAxisDP[InternalPosFig.Index[0]];

		//
		ELSIF ActPosHumAxisDP[1] < InternalPosFig.MinPosHumDP[1] THEN
			ActPosHumFigDP[InternalPosFig.Index[0]] := InternalPosFig.MinPosHumDP[1] + InternalPosFig.DispAxisDP[InternalPosFig.Index[0]];

		//
		ELSE
			ActPosHumFigDP[InternalPosFig.Index[0]] := 	InternalPosFig.CurrentPosition[InternalPosFig.Index[0]];
		END_IF

	END_FOR;

	FOR InternalPosFig.Index[1] := 3 TO 7 DO
		// Set the value at position of Middle Defender Axis by the Actual Position of Axis with Displacement of Axis
		IF (ActPosHumAxisDP[2] < InternalPosFig.MaxPosHumDP[2]) AND (ActPosHumAxisDP[2] > InternalPosFig.MinPosHumDP[2]) THEN
			ActPosHumFigDP[InternalPosFig.Index[1]] := ActPosHumAxisDP[2] + InternalPosFig.DispAxisDP[InternalPosFig.Index[1]];
			InternalPosFig.CurrentPosition[InternalPosFig.Index[1]] := ActPosHumFigDP[InternalPosFig.Index[1]];
		//
		ELSIF ActPosHumAxisDP[2] > InternalPosFig.MaxPosHumDP[2] THEN
			ActPosHumFigDP[InternalPosFig.Index[1]] := InternalPosFig.MaxPosHumDP[2] + InternalPosFig.DispAxisDP[InternalPosFig.Index[1]];

		//
		ELSIF ActPosHumAxisDP[2] < InternalPosFig.MinPosHumDP[2] THEN
			ActPosHumFigDP[InternalPosFig.Index[1]] := InternalPosFig.MinPosHumDP[2] + InternalPosFig.DispAxisDP[InternalPosFig.Index[1]];

		//
		ELSE
			ActPosHumFigDP[InternalPosFig.Index[1]] := InternalPosFig.CurrentPosition[InternalPosFig.Index[1]];
		END_IF

	END_FOR;

	FOR InternalPosFig.Index[2] := 8 TO 10 DO
		// Set the value at position of Forward Axis by the Actual Position of Axis with Displacement of Axis
		IF (ActPosHumAxisDP[3] < InternalPosFig.MaxPosHumDP[3]) AND (ActPosHumAxisDP[3] > InternalPosFig.MinPosHumDP[3]) THEN
			ActPosHumFigDP[InternalPosFig.Index[2]] := ActPosHumAxisDP[3]+ InternalPosFig.DispAxisDP[InternalPosFig.Index[2]];
			InternalPosFig.CurrentPosition[InternalPosFig.Index[2]] := ActPosHumFigDP[InternalPosFig.Index[2]];
		//
		ELSIF ActPosHumAxisDP[3] > InternalPosFig.MaxPosHumDP[3] THEN
			ActPosHumFigDP[InternalPosFig.Index[2]] := InternalPosFig.MaxPosHumDP[3] + InternalPosFig.DispAxisDP[InternalPosFig.Index[2]];

		//
		ELSIF ActPosHumAxisDP[3] < InternalPosFig.MinPosHumDP[3] THEN
			ActPosHumFigDP[InternalPosFig.Index[2]] := InternalPosFig.MinPosHumDP[3] + InternalPosFig.DispAxisDP[InternalPosFig.Index[2]];

		//
		ELSE
			ActPosHumFigDP[InternalPosFig.Index[2]] := InternalPosFig.CurrentPosition[InternalPosFig.Index[2]];
		END_IF

	END_FOR;

END_FUNCTION_BLOCK
```

### Library Logical/Libraries/Camera (ANSIC)
Depends on: sys_lib, FileIO, asstring, AsMem

#### Camera.c
```c
#include <bur/plctypes.h>
#include <math.h>

#ifdef _DEFAULT_INCLUDES
#include <AsDefault.h>
#endif

#define NaN sqrt(-1)
#define CAM_OFFLINE_MASK 128												//1000 0000b
#define CAM_ONLINE_MASK 0xFFFFFF7F

#define CAM_USER_DATA 0x10004												//Mask for user data ack
#define CAM_FIND_WHOLE_ZONE 0xFFFFFFFF										//Mask for finding at whole playground

#define MAX_DIFF_PER 0.15													//Max diffrence between old and actual value in %

#define ABS_F(X) ((X) < (0) ? -(X) : (X)) 									//ABS funkcion
							//		  |							9800
#define X1_REF_PLGND 800.0	//(UNITS) |				   3800 6800  | 11300
#define X2_REF_PLGND 11300.0//(UNITS) |				 _____|___|___|_|_
#define X1_REF_CAM 1215.0	//(PIXELS)|				| | | O O O O | | |		SCHEME OF X AXIS
#define X2_REF_CAM 82.0		//(PIXELS)|				| | O | O O | O | |		AND PLAYGROUND WITH
 							//		  |		    	| O | O O O O | O |		DISTANCE OF PLAYERS
#define Y1_REF_PLGND 820.0	//(UNITS) |	 	  		| | O | O O | O | |		IN UNITS
#define Y2_REF_PLGND -950.0 //(UNITS) |				|_|_|_O_O_O_O_|_|_|		(10 UNITS = 1 MM)
#define Y1_REF_CAM 414.0	//(PIXELS)| 		      | |   |   |
#define Y2_REF_CAM 604.0	//(PIXELS)|			 	800 | 5300 8300
							//		  |		    	   2300

#define X_LIN_EQ_K ((X1_REF_PLGND-X2_REF_PLGND)/(X1_REF_CAM-X2_REF_CAM)) 		//Define K-parameter of line equaton for X axis
#define X_LIN_EQ_Q (X1_REF_PLGND-(X1_REF_CAM*X_LIN_EQ_K))				 		//Define Q-parameter of line equaion for X axis

#define Y_LIN_EQ_K ((Y1_REF_PLGND-Y2_REF_PLGND)/(Y1_REF_CAM-Y2_REF_CAM))		//Define K-parameter of line equaton for Y axis
#define Y_LIN_EQ_Q (Y1_REF_PLGND-(Y1_REF_CAM*Y_LIN_EQ_K))						//Define Q-parameter of line equaton for Y axis

#define X_MAX_DIFF ABS_F((X_LIN_EQ_K+X_LIN_EQ_Q)-((2*X_LIN_EQ_K)+X_LIN_EQ_Q))	//Line equation for X axis
#define Y_MAX_DIFF ABS_F((Y_LIN_EQ_K+Y_LIN_EQ_Q)-((2*Y_LIN_EQ_K)+Y_LIN_EQ_Q))	//Line equation for Y axis

void setError(struct FBCamera *inst,unsigned int status);
void initFB(struct FBCamera *inst);
void resetFB(struct FBCamera *inst);
void getRealAxes(struct FBCamera *inst);
void cleanFB(struct FBCamera *inst);
REAL RctToReal_ms (struct RTCtime_typ RTCtime);

void FBCamera(struct FBCamera *inst)
{
	if ((!inst->Enable) && (!inst->Internal.disableBit))
		cleanFB(inst);

	switch (inst->Internal.MainSwitch){										//Main switch, DISABLED FB, INITialising FB, ENABLED FB and ERROR case
		/******************************************************************/
		/*							FB is DISABLED					 	  */
		/******************************************************************/

		case DISABLED:														//FB is disabled
			if (inst->Internal.disableBit){
				cleanFB(inst);
				inst->Internal.disableBit = 1;
			}
			if (inst->Enable){												//Wait for Enable = TRUE, else do nothing
				inst->Internal.MainSwitch = ENABLED;						//Go to ENABLED case
				inst->Internal.disableBit = 0;
			}
			else
				inst->Status = ERR_FUB_ENABLE_FALSE;						//Status 65534, FB is called but not enabled
			break;

		/******************************************************************/
		/*				FB is ENABLED but Camera is not ready		 	  */
		/******************************************************************/

		case ENABLED:														//FB is enabled and working
			inst->Status = ERR_OK;											//No error in enable case
			inst->Active = 1;												//variable indicating active FB
			if (!inst->InSight.ModuleOk){									//InSight Camera is not connected properly
				inst->isCameraReady = 0;									//Bit for user that Camera is not working
				if (inst->Search)											//If user allow searching for ball, change case to ERROR because you cannot find while there is no camera
					setError(inst,ERR_CAM_NOTFOUND);						//Error, Status 65533 - camera not found
			}
			else {
				inst->isCameraReady = 1;									//Bit for user that Camera is working
				inst->Internal.MainSwitch = RUN;							//Change state to RUN
			}
			break;

		/******************************************************************/
		/*						FB and Camera are ready				 	  */
		/******************************************************************/
		case RUN:															//FB is enabled and camera communicating
			if (!(inst->InSight.ModuleOk))									//if camera is disconnected change state to ENABLE where waiting for connect
				inst->Internal.MainSwitch = ENABLED;
			if (inst->Search){
				inst->isSearching = 1;
				inst->InSight.Control_I2000_S01 &= CAM_ONLINE_MASK;			//Disable control bit for cammera offline mode
				switch (inst->Internal.ChangeZone){
					case CHANGE:
						if ((inst->InSight.Control_I2000_S01 & CAM_USER_DATA) == CAM_USER_DATA){
							if ((inst->InSight.Status_I2001_S01 & 0x10000) == 0x10000) {
								if (inst->Internal.oldState == ONE_ZONE)
									inst->Internal.ChangeZone = WHOLE_ZONE;
								else
									inst->Internal.ChangeZone = ONE_ZONE;
								inst->InSight.Control_I2000_S01 &= 0xFFFEFFFB;
							}
						}
						else inst->Internal.ChangeZone = WHOLE_ZONE;
						break;

					case ONE_ZONE:
						getRealAxes(inst);
						inst->Internal.oldState = ONE_ZONE;
						if (((isnan(inst->Results.AxisX)) || isnan(inst->Results.AxisY)) && (inst->Results.NewVal)){
							inst->Internal.ChangeZone = CHANGE;
							inst->InSight.Control_I2000_S01 |= CAM_USER_DATA;
							inst->InSight.UserData_I2021_S01 = 65535;
						}
						switch (inst->Internal.Zone){
							case ZONE1:
								strcpy(inst->MappView.ZoneString,"Zone 1");
								break;

							case ZONE2:
								strcpy(inst->MappView.ZoneString,"Zone 2");
								break;

							case ZONE3:
								strcpy(inst->MappView.ZoneString,"Zone 3");
								break;

							case ZONE4:
								strcpy(inst->MappView.ZoneString,"Zone 4");
								break;

							case ZONE5:
								strcpy(inst->MappView.ZoneString,"Zone 5");
								break;

							case ZONE6:
								strcpy(inst->MappView.ZoneString,"Zone 6");
								break;

							case ZONE7:
								strcpy(inst->MappView.ZoneString,"Zone 7");
								break;

							case ZONE8:
								strcpy(inst->MappView.ZoneString,"Zone 8");
								break;

							case WHOLE:

								break;
						}
						break;

					case WHOLE_ZONE:
						getRealAxes(inst);
						inst->Internal.Zone = WHOLE;
						inst->Internal.oldState = WHOLE_ZONE;
						strcpy(inst->MappView.ZoneString,"Whole");
						if(inst->isBallFound){
							inst->Internal.ChangeZone = CHANGE;
							inst->InSight.Control_I2000_S01 |= CAM_USER_DATA;
							if (inst->Results.AxisX > 10300){
								inst->InSight.UserData_I2021_S01 = 1;
								inst->Internal.Zone = ZONE1;}
							else if (inst->Results.AxisX > 9050){
								inst->InSight.UserData_I2021_S01 = 2;
								inst->Internal.Zone = ZONE2;}
							else if (inst->Results.AxisX > 7350){
								inst->InSight.UserData_I2021_S01 = 4;
								inst->Internal.Zone = ZONE3;}
							else if (inst->Results.AxisX > 6250){
								inst->InSight.UserData_I2021_S01 = 8;
								inst->Internal.Zone = ZONE4;}
							else if (inst->Results.AxisX > 4400){
								inst->InSight.UserData_I2021_S01 = 16;
								inst->Internal.Zone = ZONE5;}
							else if (inst->Results.AxisX > 3850){
								inst->InSight.UserData_I2021_S01 = 32;
								inst->Internal.Zone = ZONE6;}
							else if (inst->Results.AxisX > 1260){
								inst->InSight.UserData_I2021_S01 = 64;
								inst->Internal.Zone = ZONE7;}
							else if(inst->Results.AxisX > 0){
								inst->InSight.UserData_I2021_S01 = 128;
								inst->Internal.Zone = ZONE8;}
							else{
								inst->Internal.ChangeZone = WHOLE_ZONE;
								inst->InSight.Control_I2000_S01 &= 0xFFFEFFFB;
								inst->InSight.UserData_I2021_S01 = 0xFFFF;
							}
						}
						break;

				}
			}
			else{
				inst->InSight.Control_I2000_S01 |= CAM_OFFLINE_MASK;
				inst->isSearching = 0;
			}
			break;

		case ERROR:															//error case, to change state is needed error Reset variable or disable FB
			inst->Error = 1;												//Change Error variable
			inst->Internal.CameraControl.ControlSwitch = WAIT_CMD;			//Reset camera trigger state
			inst->isSearching = 0;											//FB cannot searching in error case
			if (inst->ErrorReset){											//waiting on ErrorReset
				inst->Error = 0;
				inst->Status = ERR_OK;
				resetFB(inst);
				inst->Internal.MainSwitch = ENABLED;						//change state
			}
			break;
	}

	if (inst->ErrorReset)
		resetFB(inst);

	if (inst->Error == 1)
		inst->Internal.MainSwitch = ERROR;

}

void initFB(struct FBCamera *inst)
{
	inst->Active = 0;
	inst->Error = 0;
	inst->ErrorReset = 0;
	inst->isCameraReady = 0;
	inst->isBallFound = 0;
	inst->isSearching = 0;
	inst->Search = 0;
	inst->Status = ERR_OK;
	inst->Internal.CameraControl.ControlSwitch = WAIT_CMD;
	inst->Internal.MainSwitch = DISABLED;
	inst->Internal.Search_tmp = 0;
	inst->Internal.disableBit = 1;
	inst->InSight.Control_I2000_S01 |= CAM_OFFLINE_MASK;
	memset(&inst->Results.ActTime,0,sizeof(inst->Results.ActTime));
	inst->Results.AxisXOld = NaN;
	inst->Results.AxisYOld = NaN;
	inst->InSight.Control_I2000_S01 |= CAM_USER_DATA;
	inst->InSight.UserData_I2021_S01 = 65535;
	inst->Internal.ChangeZone = CHANGE;
}

void resetFB(struct FBCamera *inst)
{
	inst->ErrorReset = 0;							//Reset error reset
	inst->Error = 0;								//Reset Error
	inst->Status = ERR_OK;
}

void cleanFB(struct FBCamera *inst)
{
	initFB(inst);
	resetFB(inst);
}

void setError(struct FBCamera *inst,unsigned int status) {
	inst->Error = 1;
	inst->Status = status;
}

void getRealAxes(struct FBCamera *inst)
{
	if (inst->Internal.SuccesCount != inst->InSight.InspectionResults_I2011_S03){
		inst->Results.NewVal = 1;
		REAL AxisXnew = ((inst->InSight.InspectionResults_I2011_S01*X_LIN_EQ_K)+X_LIN_EQ_Q);
		REAL AxisYnew = ((inst->InSight.InspectionResults_I2011_S02*Y_LIN_EQ_K)+Y_LIN_EQ_Q);

		if (((AxisXnew >= 0) && (AxisXnew < 12100)) && ((AxisYnew < 3515) && (AxisYnew > -3515))){

			if (isnan(inst->Results.AxisX) || isnan(inst->Results.AxisY)){
				inst->Results.AxisX = AxisXnew;
				inst->Results.AxisY = AxisYnew;
			}
			else if(((ABS_F(AxisXnew - (inst->Results.AxisX))) < (X_MAX_DIFF * 2)) && (((ABS_F(AxisYnew - (inst->Results.AxisY))) < (Y_MAX_DIFF * 2)))) {
				inst->Results.AxisXOld = inst->Results.AxisX = ((AxisXnew + inst->Results.AxisX)/2);
				inst->Results.AxisYOld = inst->Results.AxisY = ((AxisYnew + inst->Results.AxisY)/2);
			}
			else{
				inst->Results.AxisXOld = inst->Results.AxisX;
				inst->Results.AxisYOld = inst->Results.AxisY;
				inst->Results.AxisX = AxisXnew;
				inst->Results.AxisY = AxisYnew;
			}
			memcpy((UDINT)&inst->Results.ActTimeOld,(UDINT)&inst->Results.ActTime,sizeof(inst->Results.ActTime));
			RTC_gettime(&inst->Results.ActTime);
			inst->Results.TimeDiff_ms = ((RctToReal_ms(inst->Results.ActTime)) - (RctToReal_ms(inst->Results.ActTimeOld)));
			inst->isBallFound = 1;
			inst->Status = ERR_OK;
			inst->Internal.SuccesCount = inst->InSight.InspectionResults_I2011_S03;
		}
		else{
			inst->Status = ERR_BALL_OUTRANGE;
			inst->isBallFound = 0;
		}
	}
	else if (inst->Internal.FailCount != inst->InSight.InspectionResults_I2011_S04){
		inst->Results.NewVal = 1;
		if (!isnan(inst->Results.AxisX) || !isnan(inst->Results.AxisY)){
			inst->Results.AxisXOld = inst->Results.AxisX;
			inst->Results.AxisYOld = inst->Results.AxisY;
		}
		inst->Results.AxisX = inst->Results.AxisY = NaN;
		inst->Internal.FailCount = inst->InSight.InspectionResults_I2011_S04;
		inst->isBallFound = 0;
		memcpy((UDINT)&inst->Results.ActTimeOld,(UDINT)&inst->Results.ActTime,sizeof(inst->Results.ActTime));
		RTC_gettime(&inst->Results.ActTime);
		inst->Results.TimeDiff_ms = ((RctToReal_ms(inst->Results.ActTime)) - (RctToReal_ms(inst->Results.ActTimeOld)));
	}
	else{
		inst->isBallFound = 0;
		inst->Results.NewVal = 1;
	}
}

REAL RctToReal_ms (struct RTCtime_typ RTCtime){
	return(((REAL)RTCtime.hour*3600000)+((REAL)RTCtime.minute*60000)+((REAL)RTCtime.second*1000)+((REAL)RTCtime.millisec)+((REAL)RTCtime.microsec/1000));
}
```

#### Types.typ - Exported data types
```iecst
TYPE
	MainSwitch_enum :
		(
		DISABLED := 0,
		ENABLED := 1,
		RUN := 2,
		ERROR := 255
		);
	FTPSwitch_enum :
		(
		DEVLINK := 1,
		FILECOPY := 2,
		DEVUNLINK := 3
		);
	ControlSwitch_enum :
		(
		WAIT_CMD := 0,
		TRIGGER_RDY := 1,
		TRIGGER := 2,
		ACQ := 3,
		INSP := 4
		);
	InSight_type : 	STRUCT
		ModuleOk : BOOL;
		Control_I2000_S01 : UDINT; (*Camera control including trigger*)
		Status_I2001_S01 : UDINT;
		InspectionResults_I2011_S01 : UDINT; (*X Axis*)
		InspectionResults_I2011_S02 : UDINT; (*Y Axis*)
		InspectionResults_I2011_S03 : UDINT; (*Succes*)
		InspectionResults_I2011_S04 : UDINT; (*Fail*)
		UserData_I2021_S01 : UDINT; (*Change zone*)
	END_STRUCT;
	Internal_type : 	STRUCT
		NaN : REAL;
		CameraControl : CameraControl_type;
		MainSwitch : MainSwitch_enum;
		FTP : FTP_type;
		SuccesCount : UDINT;
		FailCount : UDINT;
		disableBit : USINT;
		Search_tmp : BOOL;
		Zone : Zone_enum;
		ChangeZone : ChangeZone_enum;
		oldState : ChangeZone_enum;
	END_STRUCT;
	Zone_enum :
		(
		ZONE1 := 0,
		ZONE2 := 1,
		ZONE3 := 2,
		ZONE4 := 3,
		ZONE5 := 4,
		ZONE6 := 5,
		ZONE7 := 6,
		ZONE8 := 7,
		WHOLE := 500
		);
	ChangeZone_enum :
		(
		CHANGE := 2,
		ONE_ZONE := 1,
		WHOLE_ZONE := 0
		);
	Results_type : 	STRUCT
		AxisX : REAL;
		AxisY : REAL;
		ActTime : RTCtime_typ;
		AxisXOld : REAL;
		AxisYOld : REAL;
		TimeDiff_ms : REAL;
		ActTimeOld : RTCtime_typ;
		NewVal : BOOL;
	END_STRUCT;
	CameraControl_type : 	STRUCT
		ControlSwitch : ControlSwitch_enum;
	END_STRUCT;
	MappView_type : 	STRUCT
		ZoneString : STRING[80];
		PicEnable : BOOL;
		Y : ARRAY[0..1000]OF INT;
		X : ARRAY[0..1000]OF INT := [11(5),0,996(0)];
		LoadImage : BOOL;
	END_STRUCT;
	FTP_type : 	STRUCT
		FileCopy_0 : FileCopy;
		DevLink_0 : DevLink;
		DevUnlink_0 : DevUnlink;
		Status : USINT;
		FTPSwitch : FTPSwitch_enum;
		pParam : STRING[200];
		handle : UDINT;
		pDevice : STRING[20];
		pDest : STRING[80];
		pSrc : STRING[80];
		pDestDev : STRING[20];
	END_STRUCT;
END_TYPE
```

#### Constants.var - Exported constants
```iecst
VAR CONSTANT
	ERR_BALL_OUTRANGE : UINT := 61125; (*Ball is out of range*)
	ERR_OK : UINT := 0;
	FB_DISABLED : UINT := 65534; (*Function block is disabled*)
	ERR_CAM_NOTFOUND : UINT := 65533; (*Camera not found*)
	ERR_FTP_NOTREADY : UINT := 62687; (*FTP not ready*)
END_VAR
```

#### Camera.fun - Exported functions and function blocks
```iecst
FUNCTION_BLOCK FBCamera
	VAR_INPUT
		Enable : BOOL;
		InSight : InSight_type;
		MappView : MappView_type;
		ErrorReset : BOOL;
		Search : BOOL;
	END_VAR
	VAR_OUTPUT
		Active : BOOL;
		Error : BOOL;
		Status : UINT;
		isCameraReady : BOOL;
		isSearching : BOOL;
		isBallFound : BOOL;
		Results : Results_type;
	END_VAR
	VAR
		Internal : Internal_type;
	END_VAR
END_FUNCTION_BLOCK
```

### Library Logical/Libraries/Bar_Light (ANSIC)
Depends on: MTBasics, brsystem
